# B&R Automation Studio project NAEUL004C00R13L518F00 (part 14)

#### Act_OptP0200ToP0204BypsInitConv.st
```iecst
ACTION Act_OptP0200ToP0204BypsInitConv:

	IF p_tyNtParamCurr.bProjBypsInitConvPrep THEN

		(*Display*)
		//Initializing Conveyor
		IF EDGEPOS(p_bOpsTravLifULInitConv) THEN
			fUIInRtStatOff(ADR(tyP0200OpsGen.tyBypsInitConv.tyLyr.uiRtStat));
			fUIInRtStatOff(ADR(tyP0201OpsTravLifter.tyBypsInitConv.tyLyr.uiRtStat));
			fUIInRtStatOff(ADR(tyP0202OpsMag1.tyBypsInitConv.tyLyr.uiRtStat));
			fUIInRtStatOff(ADR(tyP0203OpsMag2.tyBypsInitConv.tyLyr.uiRtStat));
			fUIInRtStatOff(ADR(tyP0204OpsMag3.tyBypsInitConv.tyLyr.uiRtStat));
			fUIInRtStatOff(ADR(tyP0206OpsMagConv1.tyBypsInitConv.tyLyr.uiRtStat));
			fUIInRtStatOff(ADR(tyP0207OpsMagConv2.tyBypsInitConv.tyLyr.uiRtStat));
		END_IF

		//Initializing Conveyor Done
		IF EDGENEG(p_bOpsTravLifULInitConv) THEN
			fUIInRtStatHide(ADR(tyP0200OpsGen.tyBypsInitConv.tyLyr.uiRtStat));
			fUIInRtStatHide(ADR(tyP0201OpsTravLifter.tyBypsInitConv.tyLyr.uiRtStat));
			fUIInRtStatHide(ADR(tyP0202OpsMag1.tyBypsInitConv.tyLyr.uiRtStat));
			fUIInRtStatHide(ADR(tyP0203OpsMag2.tyBypsInitConv.tyLyr.uiRtStat));
			fUIInRtStatHide(ADR(tyP0204OpsMag3.tyBypsInitConv.tyLyr.uiRtStat));
			fUIInRtStatHide(ADR(tyP0206OpsMagConv1.tyBypsInitConv.tyLyr.uiRtStat));
			fUIInRtStatHide(ADR(tyP0207OpsMagConv2.tyBypsInitConv.tyLyr.uiRtStat));

			bOpsBypsInitConv	:= FALSE;
		END_IF

		//Blinking Button
		IF tyP0200OpsGen.tyBypsInitConv.tyLyr.uiRtStat.0 = FALSE THEN

			fbBypsInitConvBlinkTm(IN := TRUE);

			IF fbBypsInitConvBlinkTm.Q THEN
				fbBypsInitConvBlinkTm(IN := FALSE);

				IF tyP0200OpsGen.tyBypsInitConv.tyBtnBypsInitConv.usiBitmapIdx = 0 THEN
					tyP0200OpsGen.tyBypsInitConv.tyBtnBypsInitConv.usiBitmapIdx			:= 1;
					tyP0201OpsTravLifter.tyBypsInitConv.tyBtnBypsInitConv.usiBitmapIdx	:= 1;
					tyP0202OpsMag1.tyBypsInitConv.tyBtnBypsInitConv.usiBitmapIdx		:= 1;
					tyP0203OpsMag2.tyBypsInitConv.tyBtnBypsInitConv.usiBitmapIdx		:= 1;
					tyP0204OpsMag3.tyBypsInitConv.tyBtnBypsInitConv.usiBitmapIdx		:= 1;
					tyP0206OpsMagConv1.tyBypsInitConv.tyBtnBypsInitConv.usiBitmapIdx	:= 1;
					tyP0207OpsMagConv2.tyBypsInitConv.tyBtnBypsInitConv.usiBitmapIdx	:= 1;
				ELSE
					tyP0200OpsGen.tyBypsInitConv.tyBtnBypsInitConv.usiBitmapIdx			:= 0;
					tyP0201OpsTravLifter.tyBypsInitConv.tyBtnBypsInitConv.usiBitmapIdx	:= 0;
					tyP0202OpsMag1.tyBypsInitConv.tyBtnBypsInitConv.usiBitmapIdx		:= 0;
					tyP0203OpsMag2.tyBypsInitConv.tyBtnBypsInitConv.usiBitmapIdx		:= 0;
					tyP0204OpsMag3.tyBypsInitConv.tyBtnBypsInitConv.usiBitmapIdx		:= 0;
					tyP0206OpsMagConv1.tyBypsInitConv.tyBtnBypsInitConv.usiBitmapIdx	:= 0;
					tyP0207OpsMagConv2.tyBypsInitConv.tyBtnBypsInitConv.usiBitmapIdx	:= 0;
				END_IF

			END_IF

		ELSE

			fbBypsInitConvBlinkTm(IN := FALSE);

			tyP0200OpsGen.tyBypsInitConv.tyBtnBypsInitConv.usiBitmapIdx			:= 0;
			tyP0201OpsTravLifter.tyBypsInitConv.tyBtnBypsInitConv.usiBitmapIdx	:= 0;
			tyP0202OpsMag1.tyBypsInitConv.tyBtnBypsInitConv.usiBitmapIdx		:= 0;
			tyP0203OpsMag2.tyBypsInitConv.tyBtnBypsInitConv.usiBitmapIdx		:= 0;
			tyP0204OpsMag3.tyBypsInitConv.tyBtnBypsInitConv.usiBitmapIdx		:= 0;
			tyP0206OpsMagConv1.tyBypsInitConv.tyBtnBypsInitConv.usiBitmapIdx	:= 0;
			tyP0207OpsMagConv2.tyBypsInitConv.tyBtnBypsInitConv.usiBitmapIdx	:= 0;

		END_IF

		(*Control*)
		IF tyP0200OpsGen.tyBypsInitConv.tyBtnBypsInitConv.bRtCompl OR tyP0201OpsTravLifter.tyBypsInitConv.tyBtnBypsInitConv.bRtCompl OR tyP0202OpsMag1.tyBypsInitConv.tyBtnBypsInitConv.bRtCompl OR tyP0203OpsMag2.tyBypsInitConv.tyBtnBypsInitConv.bRtCompl OR tyP0204OpsMag3.tyBypsInitConv.tyBtnBypsInitConv.bRtCompl THEN
			tyP0200OpsGen.tyBypsInitConv.tyBtnBypsInitConv.bRtCompl			:= FALSE;
			tyP0201OpsTravLifter.tyBypsInitConv.tyBtnBypsInitConv.bRtCompl	:= FALSE;
			tyP0202OpsMag1.tyBypsInitConv.tyBtnBypsInitConv.bRtCompl		:= FALSE;
			tyP0203OpsMag2.tyBypsInitConv.tyBtnBypsInitConv.bRtCompl		:= FALSE;
			tyP0204OpsMag3.tyBypsInitConv.tyBtnBypsInitConv.bRtCompl		:= FALSE;
			tyP0206OpsMagConv1.tyBypsInitConv.tyBtnBypsInitConv.bRtCompl	:= FALSE;
			tyP0207OpsMagConv2.tyBypsInitConv.tyBtnBypsInitConv.bRtCompl	:= FALSE;

			fUIInRtStatHide(ADR(tyP0200OpsGen.tyBypsInitConv.tyLyr.uiRtStat));
			fUIInRtStatHide(ADR(tyP0201OpsTravLifter.tyBypsInitConv.tyLyr.uiRtStat));
			fUIInRtStatHide(ADR(tyP0202OpsMag1.tyBypsInitConv.tyLyr.uiRtStat));
			fUIInRtStatHide(ADR(tyP0203OpsMag2.tyBypsInitConv.tyLyr.uiRtStat));
			fUIInRtStatHide(ADR(tyP0204OpsMag3.tyBypsInitConv.tyLyr.uiRtStat));
			fUIInRtStatHide(ADR(tyP0206OpsMagConv1.tyBypsInitConv.tyLyr.uiRtStat));
			fUIInRtStatHide(ADR(tyP0207OpsMagConv2.tyBypsInitConv.tyLyr.uiRtStat));

			bOpsBypsInitConv	:= TRUE;

		ELSIF tyP0200OpsGen.tyBypsInitConv.tyHotspotClose.bRtCompl OR tyP0201OpsTravLifter.tyBypsInitConv.tyHotspotClose.bRtCompl OR tyP0202OpsMag1.tyBypsInitConv.tyHotspotClose.bRtCompl OR tyP0203OpsMag2.tyBypsInitConv.tyHotspotClose.bRtCompl OR tyP0204OpsMag3.tyBypsInitConv.tyHotspotClose.bRtCompl THEN
			tyP0200OpsGen.tyBypsInitConv.tyHotspotClose.bRtCompl		:= FALSE;
			tyP0201OpsTravLifter.tyBypsInitConv.tyHotspotClose.bRtCompl	:= FALSE;
			tyP0202OpsMag1.tyBypsInitConv.tyHotspotClose.bRtCompl		:= FALSE;
			tyP0203OpsMag2.tyBypsInitConv.tyHotspotClose.bRtCompl		:= FALSE;
			tyP0204OpsMag3.tyBypsInitConv.tyHotspotClose.bRtCompl		:= FALSE;
			tyP0206OpsMagConv1.tyBypsInitConv.tyHotspotClose.bRtCompl	:= FALSE;
			tyP0207OpsMagConv2.tyBypsInitConv.tyHotspotClose.bRtCompl	:= FALSE;

			fUIInRtStatHide(ADR(tyP0200OpsGen.tyBypsInitConv.tyLyr.uiRtStat));
			fUIInRtStatHide(ADR(tyP0201OpsTravLifter.tyBypsInitConv.tyLyr.uiRtStat));
			fUIInRtStatHide(ADR(tyP0202OpsMag1.tyBypsInitConv.tyLyr.uiRtStat));
			fUIInRtStatHide(ADR(tyP0203OpsMag2.tyBypsInitConv.tyLyr.uiRtStat));
			fUIInRtStatHide(ADR(tyP0204OpsMag3.tyBypsInitConv.tyLyr.uiRtStat));
			fUIInRtStatHide(ADR(tyP0206OpsMagConv1.tyBypsInitConv.tyLyr.uiRtStat));
			fUIInRtStatHide(ADR(tyP0207OpsMagConv2.tyBypsInitConv.tyLyr.uiRtStat));

		END_IF

	END_IF

END_ACTION
```

#### Act_OptP0202ToP0204_P0003UnloadMag.st
```iecst
ACTION Act_OptP0202ToP0204_P0003UnloadMag:

	//Reset
	IF EDGEPOS(p_bOpsStatusStop) THEN
		bUnloadMag	:= FALSE;

		tyP0202OpsMag1.tyOps.tyBtnUnloadMag.bRtCompl	:= FALSE;
		tyP0203OpsMag2.tyOps.tyBtnUnloadMag.bRtCompl	:= FALSE;
		tyP0204OpsMag3.tyOps.tyBtnUnloadMag.bRtCompl	:= FALSE;

		tyP0003MMenu.tyMMenuBtn.tyBtnMnlUnload.bRtCompl := FALSE;

		p_tyC0008MsgBox ACCESS ADR(tyP0202OpsMag1.tyMsgBoxHide);
		p_tyC0008MsgBox ACCESS ADR(tyP0203OpsMag2.tyMsgBoxHide);
		p_tyC0008MsgBox ACCESS ADR(tyP0204OpsMag3.tyMsgBoxHide);

		p_tyC0008MsgBox ACCESS ADR(tyP0003MMenu.tyMsgBoxHide);
	END_IF

	//Control
	IF tyP0202OpsMag1.tyOps.tyBtnUnloadMag.bRtCompl = TRUE THEN

		IF bUnloadMag = FALSE THEN

			p_tyC0008MsgBox ACCESS ADR(tyP0202OpsMag1.tyMsgBoxUnloadAsk);

			IF tyP0202OpsMag1.tyMsgBoxUnloadAsk.tyBtnYes.bRtCompl = TRUE THEN
				tyP0202OpsMag1.tyMsgBoxUnloadAsk.tyBtnYes.bRtCompl	:= FALSE;
				tyP0202OpsMag1.tyMsgBoxUnloadAsk.tyBtnYes.bValue	:= FALSE;

				p_tyC0008MsgBox ACCESS ADR(tyP0202OpsMag1.tyMsgBoxHide);

				bUnloadMag	:= TRUE;

				tyP0202OpsMag1.tyOps.tyBtnUnloadMag.bRtCompl	:= FALSE;

			ELSIF tyP0202OpsMag1.tyMsgBoxUnloadAsk.tyBtnNo.bRtCompl = TRUE THEN
				tyP0202OpsMag1.tyMsgBoxUnloadAsk.tyBtnNo.bRtCompl	:= FALSE;
				tyP0202OpsMag1.tyMsgBoxUnloadAsk.tyBtnNo.bValue		:= FALSE;

				p_tyC0008MsgBox ACCESS ADR(tyP0202OpsMag1.tyMsgBoxHide);

				tyP0202OpsMag1.tyOps.tyBtnUnloadMag.bRtCompl	:= FALSE;

			END_IF

		ELSE

			p_tyC0008MsgBox ACCESS ADR(tyP0202OpsMag1.tyMsgBoxResumeAsk);

			IF tyP0202OpsMag1.tyMsgBoxResumeAsk.tyBtnYes.bRtCompl = TRUE THEN
				tyP0202OpsMag1.tyMsgBoxResumeAsk.tyBtnYes.bRtCompl	:= FALSE;
				tyP0202OpsMag1.tyMsgBoxResumeAsk.tyBtnYes.bValue	:= FALSE;

				p_tyC0008MsgBox ACCESS ADR(tyP0202OpsMag1.tyMsgBoxHide);

				bUnloadMag	:= FALSE;

				tyP0202OpsMag1.tyOps.tyBtnUnloadMag.bRtCompl	:= FALSE;

			ELSIF tyP0202OpsMag1.tyMsgBoxResumeAsk.tyBtnNo.bRtCompl = TRUE THEN
				tyP0202OpsMag1.tyMsgBoxResumeAsk.tyBtnNo.bRtCompl	:= FALSE;
				tyP0202OpsMag1.tyMsgBoxResumeAsk.tyBtnNo.bValue		:= FALSE;

				p_tyC0008MsgBox ACCESS ADR(tyP0202OpsMag1.tyMsgBoxHide);

				tyP0202OpsMag1.tyOps.tyBtnUnloadMag.bRtCompl	:= FALSE;

			END_IF

		END_IF

	ELSIF tyP0203OpsMag2.tyOps.tyBtnUnloadMag.bRtCompl = TRUE THEN

		IF bUnloadMag = FALSE THEN

			p_tyC0008MsgBox ACCESS ADR(tyP0203OpsMag2.tyMsgBoxUnloadAsk);

			IF tyP0203OpsMag2.tyMsgBoxUnloadAsk.tyBtnYes.bRtCompl = TRUE THEN
				tyP0203OpsMag2.tyMsgBoxUnloadAsk.tyBtnYes.bRtCompl	:= FALSE;
				tyP0203OpsMag2.tyMsgBoxUnloadAsk.tyBtnYes.bValue	:= FALSE;

				p_tyC0008MsgBox ACCESS ADR(tyP0203OpsMag2.tyMsgBoxHide);

				bUnloadMag	:= TRUE;

				tyP0203OpsMag2.tyOps.tyBtnUnloadMag.bRtCompl	:= FALSE;

			ELSIF tyP0203OpsMag2.tyMsgBoxUnloadAsk.tyBtnNo.bRtCompl = TRUE THEN
				tyP0203OpsMag2.tyMsgBoxUnloadAsk.tyBtnNo.bRtCompl	:= FALSE;
				tyP0203OpsMag2.tyMsgBoxUnloadAsk.tyBtnNo.bValue		:= FALSE;

				p_tyC0008MsgBox ACCESS ADR(tyP0203OpsMag2.tyMsgBoxHide);

				tyP0203OpsMag2.tyOps.tyBtnUnloadMag.bRtCompl	:= FALSE;

			END_IF

		ELSE

			p_tyC0008MsgBox ACCESS ADR(tyP0203OpsMag2.tyMsgBoxResumeAsk);

			IF tyP0203OpsMag2.tyMsgBoxResumeAsk.tyBtnYes.bRtCompl = TRUE THEN
				tyP0203OpsMag2.tyMsgBoxResumeAsk.tyBtnYes.bRtCompl	:= FALSE;
				tyP0203OpsMag2.tyMsgBoxResumeAsk.tyBtnYes.bValue	:= FALSE;

				p_tyC0008MsgBox ACCESS ADR(tyP0203OpsMag2.tyMsgBoxHide);

				bUnloadMag	:= FALSE;

				tyP0203OpsMag2.tyOps.tyBtnUnloadMag.bRtCompl	:= FALSE;

			ELSIF tyP0203OpsMag2.tyMsgBoxResumeAsk.tyBtnNo.bRtCompl = TRUE THEN
				tyP0203OpsMag2.tyMsgBoxResumeAsk.tyBtnNo.bRtCompl	:= FALSE;
				tyP0203OpsMag2.tyMsgBoxResumeAsk.tyBtnNo.bValue		:= FALSE;

				p_tyC0008MsgBox ACCESS ADR(tyP0203OpsMag2.tyMsgBoxHide);

				tyP0203OpsMag2.tyOps.tyBtnUnloadMag.bRtCompl	:= FALSE;

			END_IF

		END_IF

	ELSIF tyP0204OpsMag3.tyOps.tyBtnUnloadMag.bRtCompl = TRUE THEN

		IF bUnloadMag = FALSE THEN

			p_tyC0008MsgBox ACCESS ADR(tyP0204OpsMag3.tyMsgBoxUnloadAsk);

			IF tyP0204OpsMag3.tyMsgBoxUnloadAsk.tyBtnYes.bRtCompl = TRUE THEN
				tyP0204OpsMag3.tyMsgBoxUnloadAsk.tyBtnYes.bRtCompl	:= FALSE;
				tyP0204OpsMag3.tyMsgBoxUnloadAsk.tyBtnYes.bValue	:= FALSE;

				p_tyC0008MsgBox ACCESS ADR(tyP0204OpsMag3.tyMsgBoxHide);

				bUnloadMag	:= TRUE;

				tyP0204OpsMag3.tyOps.tyBtnUnloadMag.bRtCompl	:= FALSE;

			ELSIF tyP0204OpsMag3.tyMsgBoxUnloadAsk.tyBtnNo.bRtCompl = TRUE THEN
				tyP0204OpsMag3.tyMsgBoxUnloadAsk.tyBtnNo.bRtCompl	:= FALSE;
				tyP0204OpsMag3.tyMsgBoxUnloadAsk.tyBtnNo.bValue		:= FALSE;

				p_tyC0008MsgBox ACCESS ADR(tyP0204OpsMag3.tyMsgBoxHide);

				tyP0204OpsMag3.tyOps.tyBtnUnloadMag.bRtCompl	:= FALSE;

			END_IF

		ELSE

			p_tyC0008MsgBox ACCESS ADR(tyP0204OpsMag3.tyMsgBoxResumeAsk);

			IF tyP0204OpsMag3.tyMsgBoxResumeAsk.tyBtnYes.bRtCompl = TRUE THEN
				tyP0204OpsMag3.tyMsgBoxResumeAsk.tyBtnYes.bRtCompl	:= FALSE;
				tyP0204OpsMag3.tyMsgBoxResumeAsk.tyBtnYes.bValue	:= FALSE;

				p_tyC0008MsgBox ACCESS ADR(tyP0204OpsMag3.tyMsgBoxHide);

				bUnloadMag	:= FALSE;

				tyP0204OpsMag3.tyOps.tyBtnUnloadMag.bRtCompl	:= FALSE;

			ELSIF tyP0204OpsMag3.tyMsgBoxResumeAsk.tyBtnNo.bRtCompl = TRUE THEN
				tyP0204OpsMag3.tyMsgBoxResumeAsk.tyBtnNo.bRtCompl	:= FALSE;
				tyP0204OpsMag3.tyMsgBoxResumeAsk.tyBtnNo.bValue		:= FALSE;

				p_tyC0008MsgBox ACCESS ADR(tyP0204OpsMag3.tyMsgBoxHide);

				tyP0204OpsMag3.tyOps.tyBtnUnloadMag.bRtCompl	:= FALSE;

			END_IF

		END_IF
		////////
	ELSIF tyP0003MMenu.tyMMenuBtn.tyBtnMnlUnload.bRtCompl = TRUE THEN

		IF bUnloadMag = FALSE THEN

			p_tyC0008MsgBox ACCESS ADR(tyP0003MMenu.tyMsgBoxUnloadAsk);

			IF tyP0003MMenu.tyMsgBoxUnloadAsk.tyBtnYes.bRtCompl = TRUE THEN
				tyP0003MMenu.tyMsgBoxUnloadAsk.tyBtnYes.bRtCompl	:= FALSE;
				tyP0003MMenu.tyMsgBoxUnloadAsk.tyBtnYes.bValue	:= FALSE;

				p_tyC0008MsgBox ACCESS ADR(tyP0003MMenu.tyMsgBoxHide);

				bUnloadMag	:= TRUE;

				tyP0003MMenu.tyMMenuBtn.tyBtnMnlUnload.bRtCompl	:= FALSE;

			ELSIF tyP0003MMenu.tyMsgBoxUnloadAsk.tyBtnNo.bRtCompl = TRUE THEN
				tyP0003MMenu.tyMsgBoxUnloadAsk.tyBtnNo.bRtCompl	:= FALSE;
				tyP0003MMenu.tyMsgBoxUnloadAsk.tyBtnNo.bValue		:= FALSE;

				p_tyC0008MsgBox ACCESS ADR(tyP0003MMenu.tyMsgBoxHide);

				tyP0003MMenu.tyMMenuBtn.tyBtnMnlUnload.bRtCompl	:= FALSE;

			END_IF

		ELSE

			p_tyC0008MsgBox ACCESS ADR(tyP0003MMenu.tyMsgBoxResumeAsk);

			IF tyP0003MMenu.tyMsgBoxResumeAsk.tyBtnYes.bRtCompl = TRUE THEN
				tyP0003MMenu.tyMsgBoxResumeAsk.tyBtnYes.bRtCompl	:= FALSE;
				tyP0003MMenu.tyMsgBoxResumeAsk.tyBtnYes.bValue	:= FALSE;

				p_tyC0008MsgBox ACCESS ADR(tyP0003MMenu.tyMsgBoxHide);

				bUnloadMag	:= FALSE;

				tyP0003MMenu.tyMMenuBtn.tyBtnMnlUnload.bRtCompl	:= FALSE;

			ELSIF tyP0003MMenu.tyMsgBoxResumeAsk.tyBtnNo.bRtCompl = TRUE THEN
				tyP0003MMenu.tyMsgBoxResumeAsk.tyBtnNo.bRtCompl	:= FALSE;
				tyP0003MMenu.tyMsgBoxResumeAsk.tyBtnNo.bValue		:= FALSE;

				p_tyC0008MsgBox ACCESS ADR(tyP0003MMenu.tyMsgBoxHide);

				tyP0003MMenu.tyMMenuBtn.tyBtnMnlUnload.bRtCompl	:= FALSE;

			END_IF

		END_IF

	END_IF

	//Display
	tyP0202OpsMag1.tyOps.tyBtnUnloadMag.bRtLk	:= p_bOpsStatusStop = FALSE AND bUnloadMag AND NOT p_bOpsLifMagULUnloading;
	tyP0203OpsMag2.tyOps.tyBtnUnloadMag.bRtLk	:= p_bOpsStatusStop = FALSE AND bUnloadMag AND NOT p_bOpsLifMagULUnloading;
	tyP0204OpsMag3.tyOps.tyBtnUnloadMag.bRtLk	:= p_bOpsStatusStop = FALSE AND bUnloadMag AND NOT p_bOpsLifMagULUnloading;
	tyP0003MMenu.tyMMenuBtn.tyBtnMnlUnload.bRtLk := p_bOpsStatusStop = FALSE AND bUnloadMag AND NOT p_bOpsLifMagULUnloading;

	IF p_bOpsStatusStop = FALSE AND p_bOpsLifMagULUnloading = TRUE THEN
		tyP0202OpsMag1.tyOps.tyBtnUnloadMag.usiTxtIdx	:= 1;
		tyP0203OpsMag2.tyOps.tyBtnUnloadMag.usiTxtIdx	:= 1;
		tyP0204OpsMag3.tyOps.tyBtnUnloadMag.usiTxtIdx	:= 1;
		tyP0003MMenu.tyMMenuBtn.tyBtnMnlUnload.usiTxtIdx	:= 30;
	ELSE
		tyP0202OpsMag1.tyOps.tyBtnUnloadMag.usiTxtIdx	:= 0;
		tyP0203OpsMag2.tyOps.tyBtnUnloadMag.usiTxtIdx	:= 0;
		tyP0204OpsMag3.tyOps.tyBtnUnloadMag.usiTxtIdx	:= 0;
		tyP0003MMenu.tyMMenuBtn.tyBtnMnlUnload.usiTxtIdx	:= 5;
	END_IF

	IF p_bOpsStatusStop = FALSE AND bUnloadMag = TRUE AND p_bOpsLifMagULUnloading = TRUE THEN

		fbUnloadBlinkTm(IN := TRUE);

		IF fbUnloadBlinkTm.Q = TRUE THEN
			fbUnloadBlinkTm(IN := FALSE);

			IF tyP0202OpsMag1.tyOps.tyBitmapUnloadMag.usiValueIdx = 0 THEN
				tyP0202OpsMag1.tyOps.tyBitmapUnloadMag.usiValueIdx	:= 3;
				tyP0203OpsMag2.tyOps.tyBitmapUnloadMag.usiValueIdx	:= 3;
				tyP0204OpsMag3.tyOps.tyBitmapUnloadMag.usiValueIdx	:= 3;

				tyP0003MMenu.tyMMenuBtn.tyBtnMnlUnload.usiBitmapIdx    := 4; //Yellow
			ELSE
				tyP0202OpsMag1.tyOps.tyBitmapUnloadMag.usiValueIdx	:= 0;
				tyP0203OpsMag2.tyOps.tyBitmapUnloadMag.usiValueIdx	:= 0;
				tyP0204OpsMag3.tyOps.tyBitmapUnloadMag.usiValueIdx	:= 0;

				tyP0003MMenu.tyMMenuBtn.tyBtnMnlUnload.usiBitmapIdx    := 0; //Silver
			END_IF

		END_IF

	ELSIF p_bOpsStatusStop = FALSE AND bUnloadMag = TRUE THEN

		fbUnloadBlinkTm(IN := FALSE);

		tyP0202OpsMag1.tyOps.tyBitmapUnloadMag.usiValueIdx	:= 1;
		tyP0203OpsMag2.tyOps.tyBitmapUnloadMag.usiValueIdx	:= 1;
		tyP0204OpsMag3.tyOps.tyBitmapUnloadMag.usiValueIdx	:= 1;

		tyP0003MMenu.tyMMenuBtn.tyBtnMnlUnload.usiBitmapIdx    := 1; //Green

	ELSE

		fbUnloadBlinkTm(IN := FALSE);

		tyP0202OpsMag1.tyOps.tyBitmapUnloadMag.usiValueIdx	:= 0;
		tyP0203OpsMag2.tyOps.tyBitmapUnloadMag.usiValueIdx	:= 0;
		tyP0204OpsMag3.tyOps.tyBitmapUnloadMag.usiValueIdx	:= 0;

		tyP0003MMenu.tyMMenuBtn.tyBtnMnlUnload.usiBitmapIdx    := 0;

	END_IF

	//Mask
	IF p_tyNtParamCurr.bProjLifterMagPlatform THEN
		IF p_bOpsStatusStop
			OR (p_bOpsTravLifMov AND p_bPshrConvHvBrd AND NOT(p_bOutShutterRetracted))
			THEN //p_bOpsLifMagULLifMov

			fUIInRtStatOff(ADR(tyP0202OpsMag1.tyOps.tyBtnUnloadMag.uiMaskRtStat));
			fUIInRtStatOff(ADR(tyP0203OpsMag2.tyOps.tyBtnUnloadMag.uiMaskRtStat));
			fUIInRtStatOff(ADR(tyP0204OpsMag3.tyOps.tyBtnUnloadMag.uiMaskRtStat));
			fUIInRtStatOff(ADR(tyP0003MMenu.tyMMenuBtn.tyBtnMnlUnload.uiMaskRtStat));
		ELSE
			fUIInRtStatHide(ADR(tyP0202OpsMag1.tyOps.tyBtnUnloadMag.uiMaskRtStat));
			fUIInRtStatHide(ADR(tyP0203OpsMag2.tyOps.tyBtnUnloadMag.uiMaskRtStat));
			fUIInRtStatHide(ADR(tyP0204OpsMag3.tyOps.tyBtnUnloadMag.uiMaskRtStat));
			fUIInRtStatHide(ADR(tyP0003MMenu.tyMMenuBtn.tyBtnMnlUnload.uiMaskRtStat));
		END_IF
	END_IF
END_ACTION
```

#### Act_EntP0300Disp.st
```iecst
ACTION Act_EntP0300Disp:

	//Access Addres
	p_tyC0005Main ACCESS ADR(tyCommon.tyMain);

	p_tyC0007Notif ACCESS ADR(tyCommon.tyNotif);

	p_tyC0008MsgBox ACCESS ADR(tyP0300McInfo.tyMsgBoxHide);

	p_tyC0009Info ACCESS ADR(tyCommon.tyInfo);

	p_tyP0300McInfo ACCESS ADR(tyP0300McInfo.tyMcInfo);

	//Display
	//Machine Name
	tyP0300McInfo.tyMcInfo.tyStringMcNm.sValue	:= p_tyMcParamCurr.sMcNm;

END_ACTION
```

#### Act_EntP0400Disp.st
```iecst
ACTION Act_EntP0400Disp:

	//Access Addres
	p_tyC0005Main ACCESS ADR(tyCommon.tyMain);

	p_tyC0007Notif ACCESS ADR(tyCommon.tyNotif);

	p_tyC0008MsgBox ACCESS ADR(tyP0400ProdSel.tyMsgBoxHide);

	p_tyC0009Info ACCESS ADR(tyCommon.tyInfo);

	p_tyC0011RcpPopUp ACCESS ADR(tyP0400ProdSel.tyRcpPopUp);

	p_tyP0400ProdSel ACCESS ADR(tyP0400ProdSel.tyProdSel);
	p_tyP0400RcpDet ACCESS ADR(tyP0400ProdSel.tyRcpDet);

	//Display
	tyP0400ProdSel.tyProdSel.tyBtnSort.bRtCompl			:= FALSE;
	tyP0400ProdSel.tyProdSel.tyBtnSort.bValue			:= FALSE;
	tyP0400ProdSel.tyProdSel.tyStringSearch.bRtCompl			:= TRUE;
	fUIInRtStatHide(ADR(tyP0400ProdSel.tyRcpDet.tyLyr.uiRtStat));

	fUIInRtStatHide(ADR(tyP0400ProdSel.tyRcpPopUp.tyLyr.uiRtStat)); // Hide Pop Up Layer

	//Long Board
	tyP0400ProdSel.tyProdSel.tyBtnLongBrd.uiRtStat.0			:= NOT(p_tyNtParamCurr.bProjLongBrdPrep AND p_tyMcParamCurr.bLongBrdEn);
	tyP0400ProdSel.tyRcpDet.tyBtnLongBrd.uiRtStat.0				:= NOT(p_tyNtParamCurr.bProjLongBrdPrep AND p_tyMcParamCurr.bLongBrdEn);

	//Gap Between Board
	tyP0400ProdSel.tyProdSel.tyBtnGapBetBrds.uiRtStat.0			:= NOT p_tyMcParamCurr.bGapBwtnBrdEn;
	tyP0400ProdSel.tyRcpDet.tyBtnGapBetBrd.uiRtStat.0			:= NOT p_tyMcParamCurr.bGapBwtnBrdEn;

	//Oven Info
	tyP0400ProdSel.tyProdSel.tyNumMinReqFreeBffr.uiRtStat.0		:= NOT(p_tyNtParamCurr.bOvenInfoPrep AND NOT(p_tyNtParamCurr.bOvenInfoExtdPrep AND p_tyMcParamCurr.bExtdOvenEn));
	tyP0400ProdSel.tyProdSel.tyTxtMinReqFreeBffr.uiRtStat.0		:= NOT(p_tyNtParamCurr.bOvenInfoPrep AND NOT(p_tyNtParamCurr.bOvenInfoExtdPrep AND p_tyMcParamCurr.bExtdOvenEn));
	tyP0400ProdSel.tyRcpDet.tyNumMinReqFreeBffr.uiRtStat.0		:= NOT(p_tyNtParamCurr.bOvenInfoPrep AND NOT(p_tyNtParamCurr.bOvenInfoExtdPrep AND p_tyMcParamCurr.bExtdOvenEn));
	tyP0400ProdSel.tyRcpDet.tyTxtMinReqFreeBffr.uiRtStat.0		:= NOT(p_tyNtParamCurr.bOvenInfoPrep AND NOT(p_tyNtParamCurr.bOvenInfoExtdPrep AND p_tyMcParamCurr.bExtdOvenEn));

	//Product Selection
	tyP0400ProdSel.tyProdSel.tyStringRecipeNm.sValue			:= p_tyProdRcpCurrRcp0.sRcpNm;
	tyP0400ProdSel.tyProdSel.tyNumProdWidth.diValue				:= p_tyProdRcpCurrRcp0.diWidthInUM;
	tyP0400ProdSel.tyProdSel.tyNumMaxSlt.diValue				:= p_tyProdRcpCurrRcp0.diMaxSltValue;
	tyP0400ProdSel.tyProdSel.tyNumMinSlt.diValue				:= p_tyProdRcpCurrRcp0.diMinSltValue;
	tyP0400ProdSel.tyProdSel.tyNumPitch.diValue					:= p_tyProdRcpCurrRcp0.diPitch;
	tyP0400ProdSel.tyProdSel.tyNumBrdPerSlt.diValue				:= p_tyProdRcpCurrRcp0.diBrdPerSlt;
	tyP0400ProdSel.tyProdSel.tyBtnToptoBtm.bValue				:= p_tyProdRcpCurrRcp0.bTopToBtm;
	tyP0400ProdSel.tyProdSel.tyBtnGapBetBrds.bValue				:= p_tyProdRcpCurrRcp0.bGapBwtnBrd;
	tyP0400ProdSel.tyProdSel.tyBtnLongBrd.bValue				:= p_tyProdRcpCurrRcp0.bLongBrd;
	tyP0400ProdSel.tyProdSel.tyTxtMcMode.usiValueIdx			:= p_tyProdRcpCurrRcp0.usiMcMod;
	tyP0400ProdSel.tyProdSel.tyNumMinReqFreeBffr.diValue		:= p_tyProdRcpCurrRcp0.diMinReqFreeBffr;
	tyP0400ProdSel.tyProdSel.tyNumProdWidth2.diValue			:= p_tyProdRcpCurrRcp0.diWidthInUM2;
	tyP0400ProdSel.tyProdSel.tyNumMtrPshrExtSpd.diValue			:= p_tyProdRcpCurrRcp0.diMtrPshrExtSpd;
	tyP0400ProdSel.tyProdSel.tyNumMtrPshrExtTorq.diValue		:= p_tyProdRcpCurrRcp0.diMtrPshrExtTorq;
	tyP0400ProdSel.tyProdSel.tyNumPshrOffset.diValue			:= p_tyProdRcpCurrRcp0.diPshrOffset;

END_ACTION
```

#### Act_OptP0400Search.st
```iecst
ACTION Act_OptP0400Search:

	IF tyP0400ProdSel.tyProdSel.tyStringSearch.bRtCompl = TRUE THEN	//Search Input Valid
		IF tyP0400ProdSel.tyProdSel.tyStringSearch.sValue = '' THEN
			FOR i := 1 TO c_uiP0400TableSize DO
				tyP0400ProdSel.tyProdSel.tyTableRecipe.a_tyStringDataCol0[i].sValue	:= UINT_TO_STRING(tyP0400Table.uiTablePos + i - 1);
				tyP0400ProdSel.tyProdSel.tyTableRecipe.a_tyStringDataCol1[i].sValue	:= p_tyProdRcpCurrList[tyP0400Table.uiTablePos + i - 1].sRcpNm;
				tyP0400ProdSel.tyProdSel.tyTableRecipe.a_tyStringDataCol2[i].sValue	:= p_tyProdRcpCurrList[tyP0400Table.uiTablePos + i - 1].sDisplayInfo;
			END_FOR

			tyP0400ProdSel.tyProdSel.tyStringSearch.bRtCompl	:= FALSE;

			IF tyP0400ProdSel.tyProdSel.tyBtnSort.bValue THEN
				bFilterSortP0400	:= TRUE;
			END_IF

		ELSE
			//Mask
			tyP0400ProdSel.tyProdSel.tyTableRecipe.uiMaskRtStat.0	:= FALSE;

			sProdRcpSearch	:= tyP0400ProdSel.tyProdSel.tyStringSearch.sValue;

			eProdRcpAct	:= ProdRcpActFilter;

			IF p_eProdRcpStat = ProdRcpActFilter AND p_eProdRcpStatus = Done THEN
				eProdRcpAct		:= ProdRcpActIdle;

				FOR i := 1 TO c_uiP1040TableSize DO
					tyP0400ProdSel.tyProdSel.tyTableRecipe.a_tyStringDataCol0[i].sValue	:= UINT_TO_STRING(tyP0400Table.uiTablePos + i - 1);
					tyP0400ProdSel.tyProdSel.tyTableRecipe.a_tyStringDataCol1[i].sValue	:= p_tyProdRcpFilterList[tyP0400Table.uiTablePos + i - 1].sRcpNm;
					tyP0400ProdSel.tyProdSel.tyTableRecipe.a_tyStringDataCol2[i].sValue	:= p_tyProdRcpFilterList[tyP0400Table.uiTablePos + i - 1].sDisplayInfo;
				END_FOR

				//Unmask
				tyP0400ProdSel.tyProdSel.tyTableRecipe.uiMaskRtStat.0	:= TRUE;

				tyP0400ProdSel.tyProdSel.tyStringSearch.bRtCompl		:= FALSE;

				IF tyP0400ProdSel.tyProdSel.tyBtnSort.bValue THEN
					bFilterSortP0400	:= TRUE;
				END_IF

			ELSIF p_eProdRcpStatus = Error THEN
				FOR i := 1 TO c_uiP0400TableSize DO
					tyP0400ProdSel.tyProdSel.tyTableRecipe.a_tyStringDataCol0[i].sValue		:= UINT_TO_STRING(tyP0400Table.uiTablePos + i - 1);
					tyP0400ProdSel.tyProdSel.tyTableRecipe.a_tyStringDataCol1[i].sValue		:= '';
					tyP0400ProdSel.tyProdSel.tyTableRecipe.a_tyStringDataCol2[i].sValue		:= '';
				END_FOR

				p_tyC0008MsgBox ACCESS ADR (tyP0400ProdSel.tyMsgBoxListErr);

				IF tyP0400ProdSel.tyMsgBoxListErr.tyBtnNo.bRtCompl = TRUE THEN
					tyP0400ProdSel.tyMsgBoxListErr.tyBtnNo.bRtCompl 		:= TRUE;
					tyP0400ProdSel.tyMsgBoxListErr.tyBtnNo.bValue			:= TRUE;

					p_tyC0008MsgBox ACCESS ADR (tyP0400ProdSel.tyMsgBoxHide);

					//Unmask
					tyP0400ProdSel.tyProdSel.tyTableRecipe.uiMaskRtStat.0	:= TRUE;

					//Reset
					tyP0400ProdSel.tyProdSel.tyStringSearch.bRtCompl		:= FALSE;
				END_IF
			END_IF
		END_IF
	END_IF

END_ACTION
```

#### Act_OptP0400Load.st
```iecst
ACTION Act_OptP0400Load:

	IF tyP0400ProdSel.tyProdSel.tyBtnLoad.bRtCompl = TRUE THEN

		IF usiSelProdRcpStep = 0 THEN
			//Message Confirmation Ask - Load Product Recipe
			//Mask
			tyP0400ProdSel.tyProdSel.tyTableRecipe.uiMaskRtStat		:= FALSE;
			tyP0400ProdSel.tyProdSel.tyStringSearch.uiMaskRtStat	:= FALSE;

			p_tyC0008MsgBox ACCESS ADR(tyP0400ProdSel.tyMsgBoxSelRcpAsk);

			IF tyP0400ProdSel.tyMsgBoxSelRcpAsk.tyBtnYes.bRtCompl = TRUE THEN
				tyP0400ProdSel.tyMsgBoxSelRcpAsk.tyBtnYes.bRtCompl	:= FALSE;
				tyP0400ProdSel.tyMsgBoxSelRcpAsk.tyBtnYes.bValue	:= FALSE;

				p_tyC0008MsgBox ACCESS ADR(tyP0400ProdSel.tyMsgBoxHide);

				usiSelProdRcpStep	:= 1;

			ELSIF tyP0400ProdSel.tyMsgBoxSelRcpAsk.tyBtnNo.bRtCompl = TRUE THEN
				tyP0400ProdSel.tyMsgBoxSelRcpAsk.tyBtnNo.bRtCompl	:= FALSE;
				tyP0400ProdSel.tyMsgBoxSelRcpAsk.tyBtnNo.bValue		:= FALSE;

				p_tyC0008MsgBox ACCESS ADR(tyP0400ProdSel.tyMsgBoxHide);

				usiSelProdRcpStep	:= 99;

			END_IF

		ELSIF usiSelProdRcpStep = 1 THEN
			//Load Product Recipe
			tyProdRcpInfoIn.sRcpNm		:= tyP0400ProdSel.tyProdSel.tyTableRecipe.a_tyStringDataCol1[tyP0400Table.uiSelectedRow].sValue;

			eProdRcpAct					:= ProdRcpActLoadRcp;

			IF p_eProdRcpStat = ProdRcpActLoadRcp AND p_eProdRcpStatus = Done THEN
				eProdRcpAct				:= ProdRcpActIdle;

				IF p_bProdRcpNmEmpty = TRUE AND p_bProdRcpNmNotExist = TRUE THEN
					usiSelProdRcpStep	:= 2;
				ELSE
					//Update UI Current Recipe
					tyP0400ProdSel.tyProdSel.tyStringRecipeNm.sValue		:= p_tyProdRcpCurrRcp0.sRcpNm;
					tyP0400ProdSel.tyProdSel.tyNumProdWidth.diValue			:= p_tyProdRcpCurrRcp0.diWidthInUM;
					tyP0400ProdSel.tyProdSel.tyNumMinSlt.diValue			:= p_tyProdRcpCurrRcp0.diMinSltValue;
					tyP0400ProdSel.tyProdSel.tyNumMaxSlt.diValue			:= p_tyProdRcpCurrRcp0.diMaxSltValue;
					tyP0400ProdSel.tyProdSel.tyNumPitch.diValue				:= p_tyProdRcpCurrRcp0.diPitch;
					tyP0400ProdSel.tyProdSel.tyBtnToptoBtm.bValue			:= p_tyProdRcpCurrRcp0.bTopToBtm;
					tyP0400ProdSel.tyProdSel.tyBtnGapBetBrds.bValue			:= p_tyProdRcpCurrRcp0.bGapBwtnBrd;
					tyP0400ProdSel.tyProdSel.tyBtnLongBrd.bValue			:= p_tyProdRcpCurrRcp0.bLongBrd;
					tyP0400ProdSel.tyProdSel.tyNumBrdPerSlt.diValue			:= p_tyProdRcpCurrRcp0.diBrdPerSlt;
					tyP0400ProdSel.tyProdSel.tyTxtMcMode.usiValueIdx		:= p_tyProdRcpCurrRcp0.usiMcMod;
					tyP0400ProdSel.tyProdSel.tyNumMinReqFreeBffr.diValue	:= p_tyProdRcpCurrRcp0.diMinReqFreeBffr;
					tyP0400ProdSel.tyProdSel.tyNumProdWidth2.diValue		:= p_tyProdRcpCurrRcp0.diWidthInUM2;
					tyP0400ProdSel.tyProdSel.tyNumMtrPshrExtSpd.diValue		:= p_tyProdRcpCurrRcp0.diMtrPshrExtSpd;
					tyP0400ProdSel.tyProdSel.tyNumMtrPshrExtTorq.diValue	:= p_tyProdRcpCurrRcp0.diMtrPshrExtTorq;
					tyP0400ProdSel.tyProdSel.tyNumPshrOffset.diValue		:= p_tyProdRcpCurrRcp0.diPshrOffset;

					tyProdRcpCurrRcpWr	:= p_tyProdRcpCurrRcp0;

					IF ((NOT p_tyNtParamCurr.bLFUsrSetPrep AND p_tyNtParamCurr.bLeaderMc) OR (p_tyNtParamCurr.bLFUsrSetPrep AND p_tyMcParamCurr.bLFLeaderMc)) AND p_tyNtParamCurr.bLFPrep AND p_tyMcParamCurr.bLFEn AND p_tyUsrMgmtCurrAccessRgt.bLFCtrl THEN
						usiSelProdRcpStep	:= 98;
					ELSE
						usiSelProdRcpStep	:= 99;
					END_IF

				END_IF

			ELSIF p_eProdRcpStatus = Error THEN

				usiSelProdRcpStep	:= 99;

			END_IF

		ELSIF usiSelProdRcpStep = 2 THEN
			//Message Name Not Found
			p_tyC0008MsgBox ACCESS ADR(tyP0400ProdSel.tyMsgBoxSelRcpNoNm);

			IF tyP0400ProdSel.tyMsgBoxSelRcpNoNm.tyBtnNo.bRtCompl = TRUE THEN
				tyP0400ProdSel.tyMsgBoxSelRcpNoNm.tyBtnNo.bRtCompl	:= FALSE;
				tyP0400ProdSel.tyMsgBoxSelRcpNoNm.tyBtnNo.bValue	:= FALSE;

				p_tyC0008MsgBox ACCESS ADR(tyP0400ProdSel.tyMsgBoxHide);

				usiSelProdRcpStep	:= 99;

			END_IF

		ELSIF usiSelProdRcpStep = 98 THEN
			//Message Confirmation Ask - Go To Leader Follower Control Page
			p_tyC0008MsgBox ACCESS ADR(tyP0400ProdSel.tyMsgBoxGoToLFCtrlAsk);

			IF tyP0400ProdSel.tyMsgBoxGoToLFCtrlAsk.tyBtnYes.bRtCompl = TRUE THEN
				tyP0400ProdSel.tyMsgBoxGoToLFCtrlAsk.tyBtnYes.bRtCompl	:= FALSE;
				tyP0400ProdSel.tyMsgBoxGoToLFCtrlAsk.tyBtnYes.bValue	:= FALSE;

				p_tyC0008MsgBox ACCESS ADR(tyP0400ProdSel.tyMsgBoxHide);

				eChgPage	:= UIP0700LFCtrl;

				tyCommon.tyMain.tyBtnStart.bRtCompl	:= TRUE;

				//Complete
				//Unmask
				tyP0400ProdSel.tyProdSel.tyTableRecipe.uiMaskRtStat		:= TRUE;
				tyP0400ProdSel.tyProdSel.tyStringSearch.uiMaskRtStat	:= TRUE;

				//Reset
				tyP0400ProdSel.tyProdSel.tyBtnLoad.bRtCompl	:= FALSE;
				tyP0400ProdSel.tyProdSel.tyBtnLoad.bValue	:= FALSE;

				usiSelProdRcpStep	:= 0;

			ELSIF tyP0400ProdSel.tyMsgBoxGoToLFCtrlAsk.tyBtnNo.bRtCompl = TRUE THEN
				tyP0400ProdSel.tyMsgBoxGoToLFCtrlAsk.tyBtnNo.bRtCompl	:= FALSE;
				tyP0400ProdSel.tyMsgBoxGoToLFCtrlAsk.tyBtnNo.bValue		:= FALSE;

				p_tyC0008MsgBox ACCESS ADR(tyP0400ProdSel.tyMsgBoxHide);

				usiSelProdRcpStep	:= 99;

			END_IF

		ELSIF usiSelProdRcpStep = 99 THEN
			//Complete
			//Unmask
			tyP0400ProdSel.tyProdSel.tyTableRecipe.uiMaskRtStat		:= TRUE;
			tyP0400ProdSel.tyProdSel.tyStringSearch.uiMaskRtStat	:= TRUE;

			//Reset
			tyP0400ProdSel.tyProdSel.tyBtnLoad.bRtCompl				:= FALSE;
			tyP0400ProdSel.tyProdSel.tyBtnLoad.bValue				:= FALSE;

			usiSelProdRcpStep	:= 0;

		END_IF

	END_IF

END_ACTION
```

#### Act_OptP0400Preview.st
```iecst
ACTION Act_OptP0400Preview:

	IF tyP0400ProdSel.tyProdSel.tyBtnPreview.bRtCompl = TRUE THEN

		tyProdRcpInfoIn.sRcpNm	:= tyP0400ProdSel.tyProdSel.tyTableRecipe.a_tyStringDataCol1[tyP0400Table.uiSelectedRow].sValue;

		eProdRcpAct	:= ProdRcpActGetInfo;

		IF	p_eProdRcpStat = ProdRcpActGetInfo AND p_eProdRcpStatus = Done THEN
			eProdRcpAct	:= ProdRcpActIdle;

			IF p_bProdRcpNmEmpty = TRUE AND p_bProdRcpNmNotExist = TRUE THEN
				tyP0400ProdSel.tyRcpDet.tyStringRecipeNm.sValue			:= '';
				tyP0400ProdSel.tyRcpDet.tyNumProdWidth.diValue			:= 100000;
				tyP0400ProdSel.tyRcpDet.tyNumProdWidth2.diValue			:= 100000;
				tyP0400ProdSel.tyRcpDet.tyTxtMcMode.usiValueIdx			:= p_tyMcParamCurr.usiDefaultMcMod;
				tyP0400ProdSel.tyRcpDet.tyNumFirstSlt.diValue			:= 0;
				tyP0400ProdSel.tyRcpDet.tyNumLastSlt.diValue			:= 0;
				tyP0400ProdSel.tyRcpDet.tyNumPitch.diValue				:= 0;
				tyP0400ProdSel.tyRcpDet.tyNumBrdPerSlt.diValue			:= 0;
				tyP0400ProdSel.tyRcpDet.tyBtnToptoBtm.bValue			:= FALSE;
				tyP0400ProdSel.tyRcpDet.tyBtnGapBetBrd.bValue			:= FALSE;
				tyP0400ProdSel.tyRcpDet.tyBtnLongBrd.bValue				:= FALSE;
				tyP0400ProdSel.tyRcpDet.tyNumMinReqFreeBffr.diValue		:= 0;
				tyP0400ProdSel.tyRcpDet.tyNumMtrPshrExtSpd.diValue		:= 0;
				tyP0400ProdSel.tyRcpDet.tyNumMtrPshrExtTorq.diValue		:= 0;
				tyP0400ProdSel.tyRcpDet.tyNumPshrOffset.diValue			:= p_tyProdRcpInfoOut.diPshrOffset;
			ELSE
				tyP0400ProdSel.tyRcpDet.tyStringRecipeNm.sValue			:= p_tyProdRcpInfoOut.sRcpNm;
				tyP0400ProdSel.tyRcpDet.tyNumProdWidth.diValue			:= p_tyProdRcpInfoOut.diWidthInUM;
				tyP0400ProdSel.tyRcpDet.tyNumProdWidth2.diValue			:= p_tyProdRcpInfoOut.diWidthInUM2;
				tyP0400ProdSel.tyRcpDet.tyTxtMcMode.usiValueIdx			:= p_tyProdRcpInfoOut.usiMcMod;
				tyP0400ProdSel.tyRcpDet.tyNumFirstSlt.diValue			:= p_tyProdRcpInfoOut.diMinSltValue;
				tyP0400ProdSel.tyRcpDet.tyNumLastSlt.diValue			:= p_tyProdRcpInfoOut.diMaxSltValue;
				tyP0400ProdSel.tyRcpDet.tyNumPitch.diValue				:= p_tyProdRcpInfoOut.diPitch;
				tyP0400ProdSel.tyRcpDet.tyNumBrdPerSlt.diValue			:= p_tyProdRcpInfoOut.diBrdPerSlt;
				tyP0400ProdSel.tyRcpDet.tyBtnToptoBtm.bValue			:= p_tyProdRcpInfoOut.bTopToBtm;
				tyP0400ProdSel.tyRcpDet.tyBtnGapBetBrd.bValue			:= p_tyProdRcpInfoOut.bGapBwtnBrd;
				tyP0400ProdSel.tyRcpDet.tyBtnLongBrd.bValue				:= p_tyProdRcpInfoOut.bLongBrd;
				tyP0400ProdSel.tyRcpDet.tyNumMinReqFreeBffr.diValue		:= p_tyProdRcpInfoOut.diMinReqFreeBffr;
				tyP0400ProdSel.tyRcpDet.tyNumMtrPshrExtSpd.diValue		:= p_tyProdRcpInfoOut.diMtrPshrExtSpd;
				tyP0400ProdSel.tyRcpDet.tyNumMtrPshrExtTorq.diValue		:= p_tyProdRcpInfoOut.diMtrPshrExtTorq;
				tyP0400ProdSel.tyRcpDet.tyNumPshrOffset.diValue			:= p_tyProdRcpInfoOut.diPshrOffset;
			END_IF

			fUIInRtStatOff(ADR(tyP0400ProdSel.tyRcpDet.tyLyr.uiRtStat));
			tyP0400ProdSel.tyProdSel.tyBtnPreview.bRtCompl	:= FALSE;

		END_IF

	END_IF

	IF tyP0400ProdSel.tyRcpDet.tyHotspotClose.bRtCompl = TRUE THEN
		tyP0400ProdSel.tyRcpDet.tyHotspotClose.bRtCompl	:= FALSE;
		tyP0400ProdSel.tyProdSel.tyBtnPreview.bValue	:= FALSE;

		//Hide Recipe Details
		fUIInRtStatHide(ADR(tyP0400ProdSel.tyRcpDet.tyLyr.uiRtStat));
	END_IF

	//254 Characters are Shown
	IF tyP0400ProdSel.tyRcpDet.tyHotspotShowLRcp.bRtCompl = TRUE THEN
		tyP0400ProdSel.tyRcpDet.tyHotspotShowLRcp.bRtCompl  := FALSE;

		fUIInRtStatOff(ADR(tyP0400ProdSel.tyRcpPopUp.tyLyr.uiRtStat));

		tyP0400ProdSel.tyRcpPopUp.tyStringInfo.sValue  :=  tyP0400ProdSel.tyProdSel.tyTableRecipe.a_tyStringDataCol1[tyP0400Table.uiSelectedRow].sValue; // Show 254 Characters

	ELSIF tyP0400ProdSel.tyRcpPopUp.tyHotspotClose.bRtCompl = TRUE THEN
		tyP0400ProdSel.tyRcpPopUp.tyHotspotClose.bRtCompl := FALSE;

		fUIInRtStatHide(ADR(tyP0400ProdSel.tyRcpPopUp.tyLyr.uiRtStat)); // Hide Pop Up Again

	END_IF

END_ACTION
```

#### Act_OptP0400Table.st
```iecst
ACTION Act_OptP0400Table:

	//Call Table FB
	fbP0400Table.sVisuNm			:= tyP0400Table.sVisuNm;
	fbP0400Table.udiWorkAreaStartX	:= 349;
	fbP0400Table.udiWorkAreaEndX	:= 768;
	fbP0400Table.udiWorkAreaStartY	:= 107;
	fbP0400Table.udiWorkAreaEndY	:= 428;
	fbP0400Table.udiMinXDist		:= 20;
	fbP0400Table.udiMinYDist		:= 20;
	fbP0400Table.uiSlideScale		:= c_uiP0400TableSize;
	fbP0400Table.iTotalData			:= UDINT_TO_INT(c_udiProdRcpMax);;
	fbP0400Table.iTotalRow			:= c_uiP0400TableSize;
	fbP0400Table(uiSliderStatus := tyP0400ProdSel.tyProdSel.tyTableRecipe.tyUISlider.uiRtStat , a_tyUIHotspot := tyP0400ProdSel.tyProdSel.tyTableRecipe.a_tyHotspot , uiTablePos := tyP0400Table.uiTablePos , iSliderPos := tyP0400ProdSel.tyProdSel.tyTableRecipe.tyUISlider.iValue);

	tyP0400Table.uiSelectedRow		:= fbP0400Table.uiSelectedRow;
	tyP0400Table.bTableActive		:= fbP0400Table.bTableActive;
	tyP0400Table.bSliderActive		:= fbP0400Table.bSliderActive;

	//Table Content
	iSelectedRowValue := STRING_TO_UINT(tyP0400ProdSel.tyProdSel.tyTableRecipe.a_tyStringDataCol0[tyP0400Table.uiSelectedRow].sValue);

	IF tyP0400Table.bTableActive = TRUE OR tyP0400Table.bSliderActive = TRUE OR bUpdateP0400Table THEN
		FOR i := 1 TO c_uiP0400TableSize DO
			IF tyP0400ProdSel.tyProdSel.tyBtnSort.bValue THEN

				tyP0400ProdSel.tyProdSel.tyTableRecipe.a_tyStringDataCol0[i].sValue	:= UINT_TO_STRING(tyP0400Table.uiTablePos + i - 1);
				tyP0400ProdSel.tyProdSel.tyTableRecipe.a_tyStringDataCol1[i].sValue	:= p_tyProdRcpSortedList[tyP0400Table.uiTablePos + i - 1].sRcpNm;
				tyP0400ProdSel.tyProdSel.tyTableRecipe.a_tyStringDataCol2[i].sValue	:= p_tyProdRcpSortedList[tyP0400Table.uiTablePos + i - 1].sDisplayInfo;

			ELSE

				IF tyP0400ProdSel.tyProdSel.tyStringSearch.sValue = '' THEN
					tyP0400ProdSel.tyProdSel.tyTableRecipe.a_tyStringDataCol0[i].sValue	:= UINT_TO_STRING(tyP0400Table.uiTablePos + i - 1);
					tyP0400ProdSel.tyProdSel.tyTableRecipe.a_tyStringDataCol1[i].sValue	:= p_tyProdRcpCurrList[tyP0400Table.uiTablePos + i - 1].sRcpNm;
					tyP0400ProdSel.tyProdSel.tyTableRecipe.a_tyStringDataCol2[i].sValue	:= p_tyProdRcpCurrList[tyP0400Table.uiTablePos + i - 1].sDisplayInfo;
				ELSE
					tyP0400ProdSel.tyProdSel.tyTableRecipe.a_tyStringDataCol0[i].sValue	:= UINT_TO_STRING(tyP0400Table.uiTablePos + i - 1);
					tyP0400ProdSel.tyProdSel.tyTableRecipe.a_tyStringDataCol1[i].sValue	:= p_tyProdRcpFilterList[tyP0400Table.uiTablePos + i - 1].sRcpNm;
					tyP0400ProdSel.tyProdSel.tyTableRecipe.a_tyStringDataCol2[i].sValue	:= p_tyProdRcpFilterList[tyP0400Table.uiTablePos + i - 1].sDisplayInfo;
				END_IF

			END_IF

		END_FOR

		IF bUpdateP0400Table THEN
			bUpdateP0400Table := FALSE;
		END_IF

	END_IF

	//Selected Row
	IF tyP0400Table.uiSelectedRow <> tyP0400Table.uiSelectedRowOld THEN
		FOR i := 1 TO c_uiP0400TableSize DO
			IF tyP0400Table.uiSelectedRow = i THEN
				tyP0400ProdSel.tyProdSel.tyTableRecipe.a_tyStringDataCol1[i].usiColor	:= 1;
				tyP0400ProdSel.tyProdSel.tyTableRecipe.a_tyStringDataCol2[i].usiColor	:= 1;
			ELSE
				tyP0400ProdSel.tyProdSel.tyTableRecipe.a_tyStringDataCol1[i].usiColor	:= 0;
				tyP0400ProdSel.tyProdSel.tyTableRecipe.a_tyStringDataCol2[i].usiColor	:= 0;
			END_IF
		END_FOR

		tyP0400Table.uiSelectedRowOld	:= tyP0400Table.uiSelectedRow;
	END_IF

END_ACTION
```

#### Act_OptP0400Keypad.st
```iecst
ACTION Act_OptP0400Keypad:

	IF fUIOutRtStatTPIsOpen(ADR(tyP0400ProdSel.tyProdSel.tyStringSearch.uiRtStat)) THEN
		tyProperty.tyKeypad.tyStringTitle.sKeypadTitle	:= tyP0400ProdSel.tyProdSel.tyStringSearch.sKeypadTitle;

	ELSE
		tyProperty.tyKeypad.tyStringTitle.sKeypadTitle	:= '';

	END_IF

END_ACTION
```

#### Act_EntP0410Disp.st
```iecst
ACTION Act_EntP0410Disp:

	//Access Addres
	p_tyC0005Main ACCESS ADR(tyCommon.tyMain);

	p_tyC0007Notif ACCESS ADR(tyCommon.tyNotif);

	p_tyC0008MsgBox ACCESS ADR(tyP0410MagSel.tyMsgBoxHide);

	p_tyC0009Info ACCESS ADR(tyCommon.tyInfo);

	p_tyP0410MagSel ACCESS ADR(tyP0410MagSel.tyMagSel);
	p_tyP0410MagDet ACCESS ADR(tyP0410MagSel.tyMagDet);

	tyP0410MagSel.tyMagSel.tyBtnSort.bValue 	:= FALSE;
	tyP0410MagSel.tyMagSel.tyBtnSort.bRtCompl 	:= FALSE;

	bRefreshMagRcpTable := TRUE;

	fUIInRtStatHide(ADR(tyP0410MagSel.tyMagDet.tyLyr.uiRtStat));

	// Enabling Display Auto Detect Magazine Mode
	tyP0410MagSel.tyMagSel.tyTxtMagModel.uiRtStat :=  NOT(p_tyNtParamCurr.bMagAutoVerifyPrep);

END_ACTION
```

#### Act_OptP0410Mask.st
```iecst
ACTION Act_OptP0410Mask:

	IF tyP0410MagSel.tyMagSel.tyBtnLoad.bRtCompl = FALSE THEN
		IF tyP0410MagSel.tyMagSel.tyTableRecipe.a_tyStringDataCol1[tyP0410Table.uiSelectedRow].sValue = '' THEN
			fUIInRtStatOff(ADR(tyP0410MagSel.tyMagSel.tyBtnLoad.uiMaskRtStat));
			fUIInRtStatOff(ADR(tyP0410MagSel.tyMagSel.tyBtnPreview.uiMaskRtStat));
		ELSE
			fUIInRtStatHide(ADR(tyP0410MagSel.tyMagSel.tyBtnLoad.uiMaskRtStat));
			fUIInRtStatHide(ADR(tyP0410MagSel.tyMagSel.tyBtnPreview.uiMaskRtStat));
		END_IF
	END_IF

	tyP0410MagSel.tyMagSel.tyBtnSort.uiMaskRtStat.0		:= (tyP0410MagSel.tyMagSel.tyTableRecipe.a_tyStringDataCol1[1].sValue <> '') AND (tyP0410MagSel.tyMagSel.tyBtnLoad.bRtCompl = FALSE);

END_ACTION
```

#### Act_OptP0410Load.st
```iecst
ACTION Act_OptP0410Load:

	IF tyP0410MagSel.tyMagSel.tyBtnLoad.bRtCompl = TRUE THEN

		IF usiSelMagRcpStep = 0 THEN
			//Message Confirmation Ask
			//Mask
			tyP0410MagSel.tyMagSel.tyTableRecipe.uiMaskRtStat.0		:= FALSE;
			tyP0410MagSel.tyMagSel.tyBtnPreview.uiMaskRtStat.0		:= FALSE;

			p_tyC0008MsgBox ACCESS ADR(tyP0410MagSel.tyMsgBoxSelRcpAsk);

			IF tyP0410MagSel.tyMsgBoxSelRcpAsk.tyBtnYes.bRtCompl = TRUE THEN
				tyP0410MagSel.tyMsgBoxSelRcpAsk.tyBtnYes.bRtCompl	:= FALSE;
				tyP0410MagSel.tyMsgBoxSelRcpAsk.tyBtnYes.bValue		:= FALSE;

				p_tyC0008MsgBox ACCESS ADR(tyP0410MagSel.tyMsgBoxHide);

				usiSelMagRcpStep		:= 1;

			ELSIF tyP0410MagSel.tyMsgBoxSelRcpAsk.tyBtnNo.bRtCompl = TRUE THEN
				tyP0410MagSel.tyMsgBoxSelRcpAsk.tyBtnNo.bRtCompl	:= FALSE;
				tyP0410MagSel.tyMsgBoxSelRcpAsk.tyBtnNo.bValue		:= FALSE;

				p_tyC0008MsgBox ACCESS ADR(tyP0410MagSel.tyMsgBoxHide);

				usiSelMagRcpStep		:= 99;

			END_IF

		ELSIF usiSelMagRcpStep = 1 THEN
			//Load Magazine Recipe
			tyMagRcpInfoIn.sRcpNm		:= tyP0410MagSel.tyMagSel.tyTableRecipe.a_tyStringDataCol1[tyP0410Table.uiSelectedRow].sValue;

			eMagRcpAct	:= MagRcpActLoadRcp;

			IF p_eMagRcpStat = MagRcpActLoadRcp AND p_eMagRcpStatus = Done THEN
				eMagRcpAct	:= MagRcpActIdle;

				IF p_bMagRcpNmEmpty = TRUE AND p_bMagRcpNmNotExist = TRUE THEN
					usiSelMagRcpStep	:= 2;
				ELSE
					//Update UI Current Recipe
					tyP0410MagSel.tyMagSel.tyStringRecipeNm.sValue			:= p_tyMagRcpCurrRcp.sRcpNm;
					tyP0410MagSel.tyMagSel.tyNumSltToSltDist.diValue		:= p_tyMagRcpCurrRcp.diSltToSltInUM;
					tyP0410MagSel.tyMagSel.tyNumMaxSlt.diValue				:= p_tyMagRcpCurrRcp.diTtlSlt;
					tyP0410MagSel.tyMagSel.tyNumLifterMag1Slt1Pos.diValue	:= p_tyMagRcpCurrRcp.diMag1Slt1PosInUM;
					tyP0410MagSel.tyMagSel.tyNumLifterMag2Slt1Pos.diValue	:= p_tyMagRcpCurrRcp.diMag2Slt1PosInUM;
					tyP0410MagSel.tyMagSel.tyNumLifterMag3Slt1Pos.diValue	:= p_tyMagRcpCurrRcp.diMag3Slt1PosInUM;
					tyP0410MagSel.tyMagSel.tyNumTravPosMag1.diValue			:= p_tyMagRcpCurrRcp.diMag1TravPosInUM;
					tyP0410MagSel.tyMagSel.tyNumTravPosMag2.diValue			:= p_tyMagRcpCurrRcp.diMag2TravPosInUM;
					tyP0410MagSel.tyMagSel.tyNumTravPosMag3.diValue			:= p_tyMagRcpCurrRcp.diMag3TravPosInUM;
					tyP0410MagSel.tyMagSel.tyTxtMagModel.usiValueIdx		:= p_tyMagRcpCurrRcp.usiMagModel;
					tyP0410MagSel.tyMagSel.tyNumMagMaxBrdWidth.diValue		:= p_tyMagRcpCurrRcp.diMagMaxBrdWidth;
					tyP0410MagSel.tyMagSel.tyBtnSafetyBar.bValue			:= p_tyMagRcpCurrRcp.bSafetyBarDisabled;
					tyP0410MagSel.tyMagSel.tyBtnMagHeightChkEn.bValue		:= p_tyMagRcpCurrRcp.bMagHeightChkEn;

					tyMagRcpCurrRcpWr	:= p_tyMagRcpCurrRcp;

					usiSelMagRcpStep	:= 99;
				END_IF

			ELSIF p_eProdRcpStatus = Error THEN

				usiSelMagRcpStep		:= 99;

			END_IF

		ELSIF usiSelMagRcpStep = 2 THEN
			//Message Name Not Found
			p_tyC0008MsgBox ACCESS ADR(tyP0410MagSel.tyMsgBoxSelRcpNoNm);

			IF tyP0410MagSel.tyMsgBoxSelRcpNoNm.tyBtnNo.bRtCompl = TRUE THEN
				tyP0410MagSel.tyMsgBoxSelRcpNoNm.tyBtnNo.bRtCompl	:= FALSE;
				tyP0410MagSel.tyMsgBoxSelRcpNoNm.tyBtnNo.bValue		:= FALSE;

				p_tyC0008MsgBox ACCESS ADR(tyP0410MagSel.tyMsgBoxHide);

				usiSelMagRcpStep		:= 99;

			END_IF

		ELSIF usiSelMagRcpStep = 99 THEN
			//Complete
			//Unmask
			tyP0410MagSel.tyMagSel.tyTableRecipe.uiMaskRtStat.0		:= TRUE;
			tyP0410MagSel.tyMagSel.tyBtnPreview.uiMaskRtStat.0		:= TRUE;

			//Reset
			tyP0410MagSel.tyMagSel.tyBtnLoad.bRtCompl				:= FALSE;
			tyP0410MagSel.tyMagSel.tyBtnLoad.bValue					:= FALSE;

			usiSelMagRcpStep			:= 0;

		END_IF

	END_IF

END_ACTION
```

#### Act_OptP0410Preview.st
```iecst
ACTION Act_OptP0410Preview:

	IF tyP0410MagSel.tyMagSel.tyBtnPreview.bRtCompl = TRUE THEN

		tyMagRcpInfoIn.sRcpNm	:= tyP0410MagSel.tyMagSel.tyTableRecipe.a_tyStringDataCol1[tyP0410Table.uiSelectedRow].sValue;

		eMagRcpAct				:= MagRcpActGetInfo;

		IF	p_eMagRcpStat = MagRcpActGetInfo AND p_eMagRcpStatus = Done THEN
			eMagRcpAct			:= MagRcpActIdle;

			IF p_bMagRcpNmEmpty = TRUE AND p_bMagRcpNmNotExist = TRUE THEN

				tyP0410MagSel.tyMagDet.tyStringRecipeNm.sValue			:= '';
				tyP0410MagSel.tyMagDet.tyNumSltToSltDist.diValue		:= 0;
				tyP0410MagSel.tyMagDet.tyNumMaxSlt.diValue				:= 0;
				tyP0410MagSel.tyMagDet.tyNumLifterMag1Slt1Pos.diValue	:= 0;
				tyP0410MagSel.tyMagDet.tyNumLifterMag2Slt1Pos.diValue	:= 0;
				tyP0410MagSel.tyMagDet.tyNumLifterMag3Slt1Pos.diValue	:= 0;
				tyP0410MagSel.tyMagDet.tyNumTravPosMag1.diValue			:= 0;
				tyP0410MagSel.tyMagDet.tyNumTravPosMag2.diValue			:= 0;
				tyP0410MagSel.tyMagDet.tyNumTravPosMag3.diValue			:= 0;
				tyP0410MagSel.tyMagDet.tyNumMagMaxBrdWidth.diValue		:= 0;
				tyP0410MagSel.tyMagDet.tyBtnSafetyBar.bValue			:= FALSE;
				tyP0410MagSel.tyMagDet.tyBtnMagHeightChkEn.bValue		:= FALSE;
			ELSE

				tyP0410MagSel.tyMagDet.tyStringRecipeNm.sValue			:= p_tyMagRcpInfoOut.sRcpNm;
				tyP0410MagSel.tyMagDet.tyNumSltToSltDist.diValue		:= p_tyMagRcpInfoOut.diSltToSltInUM;
				tyP0410MagSel.tyMagDet.tyNumMaxSlt.diValue				:= p_tyMagRcpInfoOut.diTtlSlt;
				tyP0410MagSel.tyMagDet.tyNumLifterMag1Slt1Pos.diValue	:= p_tyMagRcpInfoOut.diMag1Slt1PosInUM;
				tyP0410MagSel.tyMagDet.tyNumLifterMag2Slt1Pos.diValue	:= p_tyMagRcpInfoOut.diMag2Slt1PosInUM;
				tyP0410MagSel.tyMagDet.tyNumLifterMag3Slt1Pos.diValue	:= p_tyMagRcpInfoOut.diMag3Slt1PosInUM;
				tyP0410MagSel.tyMagDet.tyNumTravPosMag1.diValue			:= p_tyMagRcpInfoOut.diMag1TravPosInUM;
				tyP0410MagSel.tyMagDet.tyNumTravPosMag2.diValue			:= p_tyMagRcpInfoOut.diMag2TravPosInUM;
				tyP0410MagSel.tyMagDet.tyNumTravPosMag3.diValue			:= p_tyMagRcpInfoOut.diMag3TravPosInUM;
				tyP0410MagSel.tyMagDet.tyNumMagMaxBrdWidth.diValue		:= p_tyMagRcpInfoOut.diMagMaxBrdWidth;
				tyP0410MagSel.tyMagDet.tyBtnSafetyBar.bValue			:= p_tyMagRcpInfoOut.bSafetyBarDisabled;
				tyP0410MagSel.tyMagDet.tyBtnMagHeightChkEn.bValue		:= p_tyMagRcpInfoOut.bMagHeightChkEn;
			END_IF

			fUIInRtStatOff(ADR(tyP0410MagSel.tyMagDet.tyLyr.uiRtStat));

			tyP0410MagSel.tyMagSel.tyBtnPreview.bRtCompl				:= FALSE;
		END_IF

	END_IF

	IF tyP0410MagSel.tyMagDet.tyHotspotClose.bRtCompl = TRUE THEN
		tyP0410MagSel.tyMagDet.tyHotspotClose.bRtCompl					:= FALSE;
		tyP0410MagSel.tyMagSel.tyBtnPreview.bValue						:= FALSE;

		//Hide Recipe Details
		fUIInRtStatHide(ADR(tyP0410MagSel.tyMagDet.tyLyr.uiRtStat));
	END_IF

END_ACTION
```

#### Act_OptP0410Table.st
```iecst
ACTION Act_OptP0410Table:

	//Call Table FB
	fbP0410Table.sVisuNm			:= tyP0410Table.sVisuNm;
	fbP0410Table.udiWorkAreaStartX	:= 349;
	fbP0410Table.udiWorkAreaEndX	:= 768;
	fbP0410Table.udiWorkAreaStartY	:= 107;
	fbP0410Table.udiWorkAreaEndY	:= 428;
	fbP0410Table.udiMinXDist		:= 20;
	fbP0410Table.udiMinYDist		:= 20;
	fbP0410Table.uiSlideScale		:= c_uiP0410TableSize;
	fbP0410Table.iTotalData			:= UDINT_TO_INT(c_udiMagRcpMax);;
	fbP0410Table.iTotalRow			:= c_uiP0410TableSize;
	fbP0410Table(uiSliderStatus := tyP0410MagSel.tyMagSel.tyTableRecipe.tyUISlider.uiRtStat , a_tyUIHotspot := tyP0410MagSel.tyMagSel.tyTableRecipe.a_tyHotspot , uiTablePos := tyP0410Table.uiTablePos , iSliderPos := tyP0410MagSel.tyMagSel.tyTableRecipe.tyUISlider.iValue);

	tyP0410Table.uiSelectedRow		:= fbP0410Table.uiSelectedRow;
	tyP0410Table.bTableActive		:= fbP0410Table.bTableActive;
	tyP0410Table.bSliderActive		:= fbP0410Table.bSliderActive;

	//Table Content
	IF tyP0410Table.bTableActive = TRUE OR tyP0410Table.bSliderActive = TRUE OR bRefreshMagRcpTable OR bUpdateP0410Table THEN
		FOR i := 1 TO c_uiP0410TableSize DO
			IF tyP0410MagSel.tyMagSel.tyBtnSort.bValue THEN

				tyP0410MagSel.tyMagSel.tyTableRecipe.a_tyStringDataCol0[i].sValue	:= UINT_TO_STRING(tyP0410Table.uiTablePos + i - 1);
				tyP0410MagSel.tyMagSel.tyTableRecipe.a_tyStringDataCol1[i].sValue	:= p_tyMagRcpSortedList[tyP0410Table.uiTablePos + i - 1].sRcpNm;
				tyP0410MagSel.tyMagSel.tyTableRecipe.a_tyStringDataCol2[i].sValue	:= p_tyMagRcpSortedList[tyP0410Table.uiTablePos + i - 1].sDisplayInfo;

			ELSE
				tyP0410MagSel.tyMagSel.tyTableRecipe.a_tyStringDataCol0[i].sValue	    := UINT_TO_STRING(tyP0410Table.uiTablePos + i - 1);
				tyP0410MagSel.tyMagSel.tyTableRecipe.a_tyStringDataCol1[i].sValue		:= p_tyMagRcpCurrList[tyP0410Table.uiTablePos + i - 1].sRcpNm;
				tyP0410MagSel.tyMagSel.tyTableRecipe.a_tyStringDataCol2[i].sValue		:= p_tyMagRcpCurrList[tyP0410Table.uiTablePos + i - 1].sDisplayInfo;
			END_IF

		END_FOR

		IF bUpdateP0410Table THEN
			bUpdateP0410Table := FALSE;
		END_IF
	END_IF

	//Selected Row
	IF tyP0410Table.uiSelectedRow <> tyP0410Table.uiSelectedRowOld THEN
		FOR i := 1 TO c_uiP0410TableSize DO
			IF tyP0410Table.uiSelectedRow = i THEN
				tyP0410MagSel.tyMagSel.tyTableRecipe.a_tyStringDataCol1[i].usiColor	:= 1;
				tyP0410MagSel.tyMagSel.tyTableRecipe.a_tyStringDataCol2[i].usiColor	:= 1;
			ELSE
				tyP0410MagSel.tyMagSel.tyTableRecipe.a_tyStringDataCol1[i].usiColor	:= 0;
				tyP0410MagSel.tyMagSel.tyTableRecipe.a_tyStringDataCol2[i].usiColor	:= 0;
			END_IF
		END_FOR

		tyP0410Table.uiSelectedRowOld	:= tyP0410Table.uiSelectedRow;
	END_IF

END_ACTION
```

#### Act_OptP0410Sort.st
```iecst
ACTION Act_OptP0410Sort:

	IF tyP0410MagSel.tyMagSel.tyBtnSort.bValue THEN
		tyP0410MagSel.tyMagSel.tyBtnSort.usiTxtIdx 	:= 1;
	ELSE
		tyP0410MagSel.tyMagSel.tyBtnSort.usiTxtIdx 	:= 0;
	END_IF

	IF tyP0410MagSel.tyMagSel.tyBtnSort.bRtCompl THEN

		IF tyP0410MagSel.tyMagSel.tyBtnSort.bValue THEN

			tyP0410MagSel.tyMagSel.tyTableRecipe.uiMaskRtStat.0	:= FALSE;

			eMagRcpAct	:= MagRcpActSort;

			IF p_eMagRcpStat = MagRcpActSort AND p_eMagRcpStatus = Done THEN
				eMagRcpAct		:= MagRcpActIdle;

				FOR i := 1 TO c_uiP0410TableSize DO
					tyP0410MagSel.tyMagSel.tyTableRecipe.a_tyStringDataCol0[i].sValue	:= UINT_TO_STRING(tyP0400Table.uiTablePos + i - 1);
					tyP0410MagSel.tyMagSel.tyTableRecipe.a_tyStringDataCol1[i].sValue	:= p_tyMagRcpSortedList[tyP0400Table.uiTablePos + i - 1].sRcpNm;
					tyP0410MagSel.tyMagSel.tyTableRecipe.a_tyStringDataCol2[i].sValue	:= p_tyMagRcpSortedList[tyP0400Table.uiTablePos + i - 1].sDisplayInfo;
				END_FOR

				//Unmask
				tyP0410MagSel.tyMagSel.tyTableRecipe.uiMaskRtStat.0	:= TRUE;

				tyP0410MagSel.tyMagSel.tyBtnSort.bRtCompl := FALSE;

			ELSIF p_eMagRcpStatus = Error THEN
				FOR i := 1 TO c_uiP0410TableSize DO
					tyP0410MagSel.tyMagSel.tyTableRecipe.a_tyStringDataCol0[i].sValue		:= UINT_TO_STRING(tyP0410Table.uiTablePos + i - 1);
					tyP0410MagSel.tyMagSel.tyTableRecipe.a_tyStringDataCol1[i].sValue		:= '';
					tyP0410MagSel.tyMagSel.tyTableRecipe.a_tyStringDataCol2[i].sValue		:= '';
				END_FOR

				p_tyC0008MsgBox ACCESS ADR (tyP0410MagSel.tyMsgBoxListErr);

				IF tyP0410MagSel.tyMsgBoxListErr.tyBtnNo.bRtCompl = TRUE THEN
					tyP0410MagSel.tyMsgBoxListErr.tyBtnNo.bRtCompl 		:= TRUE;
					tyP0410MagSel.tyMsgBoxListErr.tyBtnNo.bValue			:= TRUE;

					p_tyC0008MsgBox ACCESS ADR (tyP0410MagSel.tyMsgBoxHide);

					//Unmask
					tyP0410MagSel.tyMagSel.tyTableRecipe.uiMaskRtStat.0	:= TRUE;

					//Reset
					tyP0410MagSel.tyMagSel.tyBtnSort.bRtCompl := FALSE;
				END_IF
			END_IF

		ELSE

			bUpdateP0410Table	:= TRUE;

			tyP0410MagSel.tyMagSel.tyBtnSort.bRtCompl := FALSE;

		END_IF

	END_IF

END_ACTION
```

#### Act_EntP0600Disp.st
```iecst
ACTION Act_EntP0600Disp:

	//Access Addres
	p_tyC0005Main ACCESS ADR(tyCommon.tyMain);

	p_tyC0007Notif ACCESS ADR(tyCommon.tyNotif);

	p_tyC0008MsgBox ACCESS ADR(tyP0600Alm.tyMsgBoxHide);

	p_tyC0009Info ACCESS ADR(tyCommon.tyInfo);

	p_tyC0010RcyMsg ACCESS ADR(tyP0600Alm.tyRcyMsgHide);

	p_tyP0600Alm ACCESS ADR(tyP0600Alm.tyAlm);

	tyP0600Alm.tyAlm.tyBtnCurr.bRtCompl := TRUE; //Default will be Current Alarm View

	//Reset
	bTeachTravPosA			:= FALSE;
	bTeachTravPosB			:= FALSE;
	bTeachLifterPosA		:= FALSE;
	bTeachLifterPosB		:= FALSE;
	bTeachLifterMag1Slt1Pos	:= FALSE;
	bTeachLifterMag2Slt1Pos	:= FALSE;
	bTeachLifterMag3Slt1Pos	:= FALSE;
	bTeachTravPosMag1		:= FALSE;
	bTeachTravPosMag2		:= FALSE;
	bTeachTravPosMag3		:= FALSE;
	bTeachLifterTopPos	:= FALSE;
	bTeachLifterBtmPos	:= FALSE;
	bTeachLifterTopPos2	:= FALSE;
	bTeachLifterBtmPos2	:= FALSE;

END_ACTION
```

#### Act_OptP0600RcyMsg.st
```iecst
ACTION Act_OptP0600RcyMsg:

	//Recovery Message
	FOR i := 1 TO c_uiP0600TableSize DO

		IF tyP0600Alm.tyAlm.a_tyHotspotAlm[i].bRtCompl = TRUE THEN
			tyP0600Alm.tyAlm.a_tyHotspotAlm[i].bRtCompl	:= FALSE;

			tyP0600Alm.tyRcyMsg.tyTxtMsg.udiValueIdx := p_tyAlarmRcyList[i];

			IF tyP0600Alm.tyRcyMsg.tyTxtMsg.udiValueIdx <> 0 AND tyP0600Alm.tyAlm.tyBtnHistory.bValue = FALSE THEN
				p_tyC0010RcyMsg ACCESS ADR(tyP0600Alm.tyRcyMsg);
			ELSE
				p_tyC0010RcyMsg ACCESS ADR(tyP0600Alm.tyRcyMsgHide);
			END_IF

		END_IF

	END_FOR

	// Close Recovery Message
	IF tyP0600Alm.tyRcyMsg.tyHotspotClose.bRtCompl THEN
		tyP0600Alm.tyRcyMsg.tyHotspotClose.bRtCompl := FALSE;

		p_tyC0010RcyMsg ACCESS ADR(tyP0600Alm.tyRcyMsgHide);
	END_IF

END_ACTION
```

#### Act_OptP0600Alm.st
```iecst
ACTION Act_OptP0600Alm:

	IF tyP0600Alm.tyAlm.tyBtnHistory.bRtCompl = TRUE THEN
		tyP0600Alm.tyAlm.tyBtnHistory.bRtCompl		:= FALSE;
		tyP0600Alm.tyAlm.tyBtnHistory.bValue		:= TRUE;
		tyP0600Alm.tyAlm.tyBtnCurr.bValue			:= FALSE;
	ELSIF tyP0600Alm.tyAlm.tyBtnCurr.bRtCompl = TRUE THEN
		tyP0600Alm.tyAlm.tyBtnCurr.bRtCompl			:= FALSE;
		tyP0600Alm.tyAlm.tyBtnCurr.bValue			:= TRUE;
		tyP0600Alm.tyAlm.tyBtnHistory.bValue		:= FALSE;
	END_IF

	IF NOT p_bAlarmErr THEN
		memset(ADR(tyUIAlmData.bAlm) , 0 , SIZEOF(tyUIAlmData.bAlm));
	END_IF

	IF NOT p_bAlarmWarning THEN
		memset(ADR(tyUIAlmData.bWarning) , 0 , SIZEOF(tyUIAlmData.bWarning));
	ELSE
		IF p_bUSHermesAConnected OR p_tyMcParamCurr.eUSCommA = McSetCommModSMEMA THEN
			tyUIAlmData.bWarning[3114] := FALSE;
		END_IF
		IF p_bUSHermesBConnected OR p_tyMcParamCurr.eUSCommB = McSetCommModSMEMA THEN
			tyUIAlmData.bWarning[3281] := FALSE;
		END_IF
	END_IF

	IF tyP0600Alm.tyAlm.tyBtnCurr.bValue = TRUE THEN

		fUIInRtStatOff(ADR(tyP0600Alm.tyAlm.tyAlarm.tyUIAlmCur.uiRtStat));
		fUIInRtStatHide(ADR(tyP0600Alm.tyAlm.tyAlarm.tyUIAlmHis.uiRtStat));
		tyP0600Alm.tyAlm.tyBtnHistoryUp.uiMaskRtStat.0 		:= FALSE;
		tyP0600Alm.tyAlm.tyBtnHistoryDown.uiMaskRtStat.0 	:= FALSE;

		FOR i := 1 TO c_uiP0600TableSize DO
			IF p_bStartupUISettingsLoadDone THEN
				IF p_tyAlarmCurrList[i].eSeverity = AlmSeverityError THEN
					tyUIAlmData.bAlm[p_tyAlarmCurrList[i].udiErrorCode] := p_tyAlarmCurrList[i].bAlm;
				ELSIF p_tyAlarmCurrList[i].eSeverity = AlmSeverityWarning THEN
					tyUIAlmData.bWarning[p_tyAlarmCurrList[i].udiErrorCode] := p_tyAlarmCurrList[i].bWarning;
				END_IF
			END_IF
		END_FOR

	ELSIF tyP0600Alm.tyAlm.tyBtnHistory.bValue = TRUE THEN

		fUIInRtStatHide(ADR(tyP0600Alm.tyAlm.tyAlarm.tyUIAlmCur.uiRtStat));
		fUIInRtStatOff(ADR(tyP0600Alm.tyAlm.tyAlarm.tyUIAlmHis.uiRtStat));
		tyP0600Alm.tyAlm.tyBtnHistoryUp.uiMaskRtStat.0 		:= TRUE;
		tyP0600Alm.tyAlm.tyBtnHistoryDown.uiMaskRtStat.0 	:= TRUE;

	END_IF

END_ACTION
```

#### Act_EntP0700Disp.st
```iecst
ACTION Act_EntP0700Disp:

	//Access Address
	p_tyC0005Main ACCESS ADR(tyCommon.tyMain);

	p_tyC0007Notif ACCESS ADR(tyCommon.tyNotif);

	p_tyC0008MsgBox ACCESS ADR(tyP0700LFCtrl.tyMsgBoxHide);

	p_tyC0009Info ACCESS ADR(tyCommon.tyInfo);

	p_tyP0700LFCtrl ACCESS ADR(tyP0700LFCtrl.tyLdr);

	//Run
	bLeaderRun	:= TRUE;

END_ACTION
```

#### Act_ExitP0700.st
```iecst
ACTION Act_ExitP0700:

	IF NOT(tyP0700LFCtrl.tyLdr.tyBtnChgAll.bRtCompl OR tyP0700LFCtrl.tyLdr.tyBtnChgSeqAuto.bRtCompl OR tyP0700LFCtrl.tyLdr.tyBtnChgSeqMnl.bRtCompl OR tyP0700LFCtrl.tyLdr.tyBtnSyncTm.bRtCompl) THEN
		bLeaderRun	:= FALSE;
		bLFRunInBG	:= FALSE;
	ELSE
		bLFRunInBG	:= TRUE;
	END_IF

	usiChgPage	:= 1;

END_ACTION
```

#### Act_OptP0700LFLeaderCtrl.st
```iecst
ACTION Act_OptP0700LFLeaderCtrl:

	CASE usiLFLeaderCtrlStep OF
		0:	//Confirmation Message - Execute Ask
			IF tyP0700LFCtrl.tyLdr.tyBtnChgAll.bRtCompl THEN

				p_tyC0008MsgBox ACCESS ADR(tyP0700LFCtrl.tyMsgBoxChgAllAsk);

				IF tyP0700LFCtrl.tyMsgBoxChgAllAsk.tyBtnYes.bRtCompl = TRUE THEN
					tyP0700LFCtrl.tyMsgBoxChgAllAsk.tyBtnYes.bRtCompl	:= FALSE;
					tyP0700LFCtrl.tyMsgBoxChgAllAsk.tyBtnYes.bValue		:= FALSE;

					p_tyC0008MsgBox ACCESS ADR(tyP0700LFCtrl.tyMsgBoxHide);

					tyP0700LFCtrl.tyLdr.tyBtnChgAll.bValue		:= TRUE;

					usiLFLeaderCtrlStep	:= 2;

				ELSIF tyP0700LFCtrl.tyMsgBoxChgAllAsk.tyBtnNo.bRtCompl = TRUE THEN
					tyP0700LFCtrl.tyMsgBoxChgAllAsk.tyBtnNo.bRtCompl	:= FALSE;
					tyP0700LFCtrl.tyMsgBoxChgAllAsk.tyBtnNo.bValue		:= FALSE;

					p_tyC0008MsgBox ACCESS ADR(tyP0700LFCtrl.tyMsgBoxHide);

					tyP0700LFCtrl.tyLdr.tyBtnChgAll.bValue		:= FALSE;
					tyP0700LFCtrl.tyLdr.tyBtnChgAll.bRtCompl	:= FALSE;

				END_IF

			ELSIF tyP0700LFCtrl.tyLdr.tyBtnChgSeqAuto.bRtCompl THEN

				p_tyC0008MsgBox ACCESS ADR(tyP0700LFCtrl.tyMsgBoxChgSeqAutoAsk);

				IF tyP0700LFCtrl.tyMsgBoxChgSeqAutoAsk.tyBtnYes.bRtCompl = TRUE THEN
					tyP0700LFCtrl.tyMsgBoxChgSeqAutoAsk.tyBtnYes.bRtCompl	:= FALSE;
					tyP0700LFCtrl.tyMsgBoxChgSeqAutoAsk.tyBtnYes.bValue		:= FALSE;

					p_tyC0008MsgBox ACCESS ADR(tyP0700LFCtrl.tyMsgBoxHide);

					tyP0700LFCtrl.tyLdr.tyBtnChgSeqAuto.bValue		:= TRUE;

					usiLFLeaderCtrlStep	:= 2;

				ELSIF tyP0700LFCtrl.tyMsgBoxChgSeqAutoAsk.tyBtnNo.bRtCompl = TRUE THEN
					tyP0700LFCtrl.tyMsgBoxChgSeqAutoAsk.tyBtnNo.bRtCompl	:= FALSE;
					tyP0700LFCtrl.tyMsgBoxChgSeqAutoAsk.tyBtnNo.bValue		:= FALSE;

					p_tyC0008MsgBox ACCESS ADR(tyP0700LFCtrl.tyMsgBoxHide);

					tyP0700LFCtrl.tyLdr.tyBtnChgSeqAuto.bValue		:= FALSE;
					tyP0700LFCtrl.tyLdr.tyBtnChgSeqAuto.bRtCompl	:= FALSE;

				END_IF

			ELSIF tyP0700LFCtrl.tyLdr.tyBtnChgSeqMnl.bRtCompl THEN

				p_tyC0008MsgBox ACCESS ADR(tyP0700LFCtrl.tyMsgBoxChgSeqMnlAsk);

				IF tyP0700LFCtrl.tyMsgBoxChgSeqMnlAsk.tyBtnYes.bRtCompl = TRUE THEN
					tyP0700LFCtrl.tyMsgBoxChgSeqMnlAsk.tyBtnYes.bRtCompl	:= FALSE;
					tyP0700LFCtrl.tyMsgBoxChgSeqMnlAsk.tyBtnYes.bValue		:= FALSE;

					p_tyC0008MsgBox ACCESS ADR(tyP0700LFCtrl.tyMsgBoxHide);

					tyP0700LFCtrl.tyLdr.tyBtnChgSeqMnl.bValue	:= TRUE;

					usiLFLeaderCtrlStep	:= 2;

				ELSIF tyP0700LFCtrl.tyMsgBoxChgSeqMnlAsk.tyBtnNo.bRtCompl = TRUE THEN
					tyP0700LFCtrl.tyMsgBoxChgSeqMnlAsk.tyBtnNo.bRtCompl		:= FALSE;
					tyP0700LFCtrl.tyMsgBoxChgSeqMnlAsk.tyBtnNo.bValue		:= FALSE;

					p_tyC0008MsgBox ACCESS ADR(tyP0700LFCtrl.tyMsgBoxHide);

					tyP0700LFCtrl.tyLdr.tyBtnChgSeqMnl.bValue	:= FALSE;
					tyP0700LFCtrl.tyLdr.tyBtnChgSeqMnl.bRtCompl	:= FALSE;

				END_IF

			ELSIF tyP0700LFCtrl.tyLdr.tyBtnSyncTm.bRtCompl THEN

				p_tyC0008MsgBox ACCESS ADR(tyP0700LFCtrl.tyMsgBoxSyncPLCTmAsk);

				IF tyP0700LFCtrl.tyMsgBoxSyncPLCTmAsk.tyBtnYes.bRtCompl = TRUE THEN
					tyP0700LFCtrl.tyMsgBoxSyncPLCTmAsk.tyBtnYes.bRtCompl	:= FALSE;
					tyP0700LFCtrl.tyMsgBoxSyncPLCTmAsk.tyBtnYes.bValue		:= FALSE;

					p_tyC0008MsgBox ACCESS ADR(tyP0700LFCtrl.tyMsgBoxHide);

					tyP0700LFCtrl.tyLdr.tyBtnSyncTm.bValue		:= TRUE;

					usiLFLeaderCtrlStep	:= 2;

				ELSIF tyP0700LFCtrl.tyMsgBoxSyncPLCTmAsk.tyBtnNo.bRtCompl = TRUE THEN
					tyP0700LFCtrl.tyMsgBoxSyncPLCTmAsk.tyBtnNo.bRtCompl		:= FALSE;
					tyP0700LFCtrl.tyMsgBoxSyncPLCTmAsk.tyBtnNo.bValue		:= FALSE;

					p_tyC0008MsgBox ACCESS ADR(tyP0700LFCtrl.tyMsgBoxHide);

					tyP0700LFCtrl.tyLdr.tyBtnSyncTm.bValue		:= FALSE;
					tyP0700LFCtrl.tyLdr.tyBtnSyncTm.bRtCompl	:= FALSE;

				END_IF

			END_IF

		1:	//Confirmation Message - Terminate Ask
			p_tyC0008MsgBox ACCESS ADR(tyP0700LFCtrl.tyMsgBoxTerminateOpsAsk);

			IF tyP0700LFCtrl.tyMsgBoxTerminateOpsAsk.tyBtnYes.bRtCompl = TRUE THEN
				tyP0700LFCtrl.tyMsgBoxTerminateOpsAsk.tyBtnYes.bRtCompl	:= FALSE;
				tyP0700LFCtrl.tyMsgBoxTerminateOpsAsk.tyBtnYes.bValue	:= FALSE;

				p_tyC0008MsgBox ACCESS ADR(tyP0700LFCtrl.tyMsgBoxHide);

				usiLFLeaderCtrlStep	:= 3;

			ELSIF tyP0700LFCtrl.tyMsgBoxTerminateOpsAsk.tyBtnNo.bRtCompl = TRUE THEN
				tyP0700LFCtrl.tyMsgBoxTerminateOpsAsk.tyBtnNo.bRtCompl	:= FALSE;
				tyP0700LFCtrl.tyMsgBoxTerminateOpsAsk.tyBtnNo.bValue	:= FALSE;

				p_tyC0008MsgBox ACCESS ADR(tyP0700LFCtrl.tyMsgBoxHide);

				tyP0700LFCtrl.tyLdr.tyBtnChgAll.bValue		:= tyP0700LFCtrl.tyLdr.tyBtnChgAll.bRtCompl;
				tyP0700LFCtrl.tyLdr.tyBtnChgSeqAuto.bValue	:= tyP0700LFCtrl.tyLdr.tyBtnChgSeqAuto.bRtCompl;
				tyP0700LFCtrl.tyLdr.tyBtnChgSeqMnl.bValue	:= tyP0700LFCtrl.tyLdr.tyBtnChgSeqMnl.bRtCompl;
				tyP0700LFCtrl.tyLdr.tyBtnSyncTm.bValue		:= tyP0700LFCtrl.tyLdr.tyBtnSyncTm.bRtCompl;

				usiLFLeaderCtrlStep	:= 2;

			END_IF

			//Display
			tyP0700LFCtrl.tyLdr.tyBitmapChgAll.usiValueIdx		:= BOOL_TO_USINT(tyP0700LFCtrl.tyLdr.tyBtnChgAll.bRtCompl);
			tyP0700LFCtrl.tyLdr.tyBitmapChgSeqAuto.usiValueIdx	:= BOOL_TO_USINT(tyP0700LFCtrl.tyLdr.tyBtnChgSeqAuto.bRtCompl);
			tyP0700LFCtrl.tyLdr.tyBitmapChgSeqMnl.usiValueIdx	:= BOOL_TO_USINT(tyP0700LFCtrl.tyLdr.tyBtnChgSeqMnl.bRtCompl);
			tyP0700LFCtrl.tyLdr.tyBitmapSyncTm.usiValueIdx		:= BOOL_TO_USINT(tyP0700LFCtrl.tyLdr.tyBtnSyncTm.bRtCompl);

		2:	//Processing
			IF tyP0700LFCtrl.tyLdr.tyBtnChgAll.bRtCompl THEN
				eLFLeaderAct	:= LFActChgAllAuto;

				IF p_eLFLeaderStat = LFActChgAllAuto AND (p_eLFLeaderStatus = Done OR p_eLFLeaderStatus = Error) THEN
					usiLFLeaderCtrlStep	:= 3;
				ELSIF tyP0700LFCtrl.tyLdr.tyBtnChgAll.bValue = FALSE THEN
					usiLFLeaderCtrlStep	:= 1;
				END_IF

			ELSIF tyP0700LFCtrl.tyLdr.tyBtnChgSeqAuto.bRtCompl THEN
				eLFLeaderAct	:= LFActChgSeqAuto;

				IF p_tyMcParamCurr.bLFSeqStayActive = FALSE THEN
					IF p_eLFLeaderStat = LFActChgSeqAuto AND (p_eLFLeaderStatus = Done OR p_eLFLeaderStatus = Error) THEN
						usiLFLeaderCtrlStep	:= 3;
					ELSIF tyP0700LFCtrl.tyLdr.tyBtnChgSeqAuto.bValue = FALSE THEN
						usiLFLeaderCtrlStep	:= 1;
					END_IF
				ELSE
					IF p_eLFLeaderStat = LFActChgSeqAuto AND p_eLFLeaderStatus = Error THEN
						usiLFLeaderCtrlStep	:= 4;
					ELSIF tyP0700LFCtrl.tyLdr.tyBtnChgSeqAuto.bValue = FALSE THEN
						usiLFLeaderCtrlStep	:= 1;
					END_IF
				END_IF

			ELSIF tyP0700LFCtrl.tyLdr.tyBtnChgSeqMnl.bRtCompl THEN
				eLFLeaderAct	:= LFActChgSeqMnl;

				IF p_tyMcParamCurr.bLFSeqStayActive = FALSE THEN
					IF p_eLFLeaderStat = LFActChgSeqMnl AND (p_eLFLeaderStatus = Done OR p_eLFLeaderStatus = Error) THEN
						usiLFLeaderCtrlStep	:= 3;
					ELSIF tyP0700LFCtrl.tyLdr.tyBtnChgSeqMnl.bValue = FALSE THEN
						usiLFLeaderCtrlStep	:= 1;
					END_IF
				ELSE
					IF p_eLFLeaderStat = LFActChgSeqMnl AND p_eLFLeaderStatus = Error THEN
						usiLFLeaderCtrlStep	:= 4;
					ELSIF tyP0700LFCtrl.tyLdr.tyBtnChgSeqMnl.bValue = FALSE THEN
						usiLFLeaderCtrlStep	:= 1;
					END_IF
				END_IF

			ELSIF tyP0700LFCtrl.tyLdr.tyBtnSyncTm.bRtCompl THEN
				eLFLeaderAct	:= LFActSyncPLCTm;

				IF p_eLFLeaderStat = LFActSyncPLCTm AND (p_eLFLeaderStatus = Done OR p_eLFLeaderStatus = Error) THEN
					usiLFLeaderCtrlStep	:= 3;
				ELSIF tyP0700LFCtrl.tyLdr.tyBtnSyncTm.bValue = FALSE THEN
					usiLFLeaderCtrlStep	:= 1;
				END_IF

			END_IF

			//Display
			fbLFLeaderCtrlBlinkTm(IN := TRUE);
			IF fbLFLeaderCtrlBlinkTm.Q = TRUE THEN
				fbLFLeaderCtrlBlinkTm(IN := FALSE);

				tyP0700LFCtrl.tyLdr.tyBitmapChgAll.usiValueIdx		:= BOOL_TO_USINT(USINT_TO_BOOL(tyP0700LFCtrl.tyLdr.tyBitmapChgAll.usiValueIdx) XOR tyP0700LFCtrl.tyLdr.tyBtnChgAll.bRtCompl);
				tyP0700LFCtrl.tyLdr.tyBitmapChgSeqAuto.usiValueIdx	:= BOOL_TO_USINT(USINT_TO_BOOL(tyP0700LFCtrl.tyLdr.tyBitmapChgSeqAuto.usiValueIdx) XOR tyP0700LFCtrl.tyLdr.tyBtnChgSeqAuto.bRtCompl);
				tyP0700LFCtrl.tyLdr.tyBitmapChgSeqMnl.usiValueIdx	:= BOOL_TO_USINT(USINT_TO_BOOL(tyP0700LFCtrl.tyLdr.tyBitmapChgSeqMnl.usiValueIdx) XOR tyP0700LFCtrl.tyLdr.tyBtnChgSeqMnl.bRtCompl);
				tyP0700LFCtrl.tyLdr.tyBitmapSyncTm.usiValueIdx		:= BOOL_TO_USINT(USINT_TO_BOOL(tyP0700LFCtrl.tyLdr.tyBitmapSyncTm.usiValueIdx) XOR tyP0700LFCtrl.tyLdr.tyBtnSyncTm.bRtCompl);
			END_IF

		3:	//Complete Reset
			usiLFLeaderCtrlStep	:= 0;

			eLFLeaderAct	:= LFActIdle;

			fbLFLeaderCtrlBlinkTm(IN := FALSE);

			tyP0700LFCtrl.tyLdr.tyBitmapChgAll.usiValueIdx		:= 0;
			tyP0700LFCtrl.tyLdr.tyBitmapChgSeqAuto.usiValueIdx	:= 0;
			tyP0700LFCtrl.tyLdr.tyBitmapChgSeqMnl.usiValueIdx	:= 0;
			tyP0700LFCtrl.tyLdr.tyBitmapSyncTm.usiValueIdx		:= 0;

			tyP0700LFCtrl.tyLdr.tyBtnChgAll.bRtCompl			:= FALSE;
			tyP0700LFCtrl.tyLdr.tyBtnChgSeqAuto.bRtCompl		:= FALSE;
			tyP0700LFCtrl.tyLdr.tyBtnChgSeqMnl.bRtCompl			:= FALSE;
			tyP0700LFCtrl.tyLdr.tyBtnSyncTm.bRtCompl			:= FALSE;

			tyP0700LFCtrl.tyLdr.tyBtnChgAll.bValue				:= FALSE;
			tyP0700LFCtrl.tyLdr.tyBtnChgSeqAuto.bValue			:= FALSE;
			tyP0700LFCtrl.tyLdr.tyBtnChgSeqMnl.bValue			:= FALSE;
			tyP0700LFCtrl.tyLdr.tyBtnSyncTm.bValue				:= FALSE;

		4:
			p_tyC0008MsgBox ACCESS ADR(tyP0700LFCtrl.tyMsgBoxErrorAsk);

			IF tyP0700LFCtrl.tyMsgBoxErrorAsk.tyBtnNo.bRtCompl = TRUE THEN
				tyP0700LFCtrl.tyMsgBoxErrorAsk.tyBtnNo.bRtCompl	:= FALSE;
				tyP0700LFCtrl.tyMsgBoxErrorAsk.tyBtnNo.bValue	:= FALSE;

				p_tyC0008MsgBox ACCESS ADR(tyP0700LFCtrl.tyMsgBoxHide);

				usiLFLeaderCtrlStep	:= 3;

			END_IF

	END_CASE

END_ACTION
```

#### Act_OptP0700Table.st
```iecst
ACTION Act_OptP0700Table:

	//Call Table FB
	fbP0700Table.sVisuNm			:= tyP0700Table.sVisuNm;
	fbP0700Table.udiWorkAreaStartX	:= 17;
	fbP0700Table.udiWorkAreaEndX	:= 594;
	fbP0700Table.udiWorkAreaStartY	:= 94;
	fbP0700Table.udiWorkAreaEndY	:= 445;
	fbP0700Table.udiMinXDist		:= 20;
	fbP0700Table.udiMinYDist		:= 20;
	fbP0700Table.uiSlideScale		:= c_uiP0700TableSize;
	fbP0700Table.iTotalData			:= UDINT_TO_INT(c_diLFClntNum);
	fbP0700Table.iTotalRow			:= c_uiP0700TableSize;
	fbP0700Table(uiSliderStatus 	:= tyP0700LFCtrl.tyLdr.tyTable1List.tyUISlider.uiRtStat , a_tyUIHotspot := tyP0700LFCtrl.tyLdr.tyTable1List.a_tyHotspot , uiTablePos := tyP0700Table.uiTablePos , iSliderPos := tyP0700LFCtrl.tyLdr.tyTable1List.tyUISlider.iValue);

	tyP0700Table.uiSelectedRow		:= fbP0700Table.uiSelectedRow;
	tyP0700Table.bTableActive		:= fbP0700Table.bTableActive;
	tyP0700Table.bSliderActive		:= fbP0700Table.bSliderActive;

	//Table Content
	IF tyP0700Table.bTableActive = TRUE OR tyP0700Table.bSliderActive = TRUE THEN
		FOR i := 1 TO c_uiP0700TableSize DO
			tyP0700LFCtrl.tyLdr.tyTable1List.a_tyStringDataCol0[i].sValue	:= UINT_TO_STRING(tyP0700Table.uiTablePos + i - 1);
		END_FOR
	END_IF

	//Update Status & Current Recipe
	FOR i := 1 TO c_uiP0700TableSize DO
		tyP0700LFCtrl.tyLdr.tyTable1List.a_tyStringDataCol1[i].sValue	:= p_tyLFLeaderFollowerToLeaderTag[tyP0700Table.uiTablePos + i - 1].sMcNm;
		tyP0700LFCtrl.tyLdr.tyTable1List.a_tyStringDataCol2[i].sValue	:= p_tyLFLeaderFollowerToLeaderTag[tyP0700Table.uiTablePos + i - 1].sIPAddr;
		tyP0700LFCtrl.tyLdr.tyTable1List.a_tyStringDataCol4[i].sValue	:= p_tyLFLeaderFollowerToLeaderTag[tyP0700Table.uiTablePos + i - 1].sCurrProdRcp;

		IF p_tyLFLeaderFollowerToLeaderTag[tyP0700Table.uiTablePos + i - 1].sIPAddr = '' THEN
			tyP0700LFCtrl.tyLdr.tyTable1List.a_tyTxtDataCol3[i].usiValueIdx	:= 0;	//Empty
		ELSIF p_tyLFLeaderFollowerToLeaderTag[tyP0700Table.uiTablePos + i - 1].sIPAddr = '0000' THEN
			tyP0700LFCtrl.tyLdr.tyTable1List.a_tyTxtDataCol3[i].usiValueIdx	:= 1;	//Third Party
		ELSIF p_tyMcParamCurr.a_bLFOnline[tyP0700Table.uiTablePos + i - 1] = FALSE THEN
			tyP0700LFCtrl.tyLdr.tyTable1List.a_tyTxtDataCol3[i].usiValueIdx	:= 2;	//Offline
		ELSIF p_tyLFLeaderFollowerToLeaderTag[tyP0700Table.uiTablePos + i - 1].sIPAddr = p_sHWInfoIPAddr THEN
			tyP0700LFCtrl.tyLdr.tyTable1List.a_tyTxtDataCol3[i].usiValueIdx	:= 4;	//Leader
		ELSIF p_tyLFLeaderFollowerToLeaderTag[tyP0700Table.uiTablePos + i - 1].bSectionLeader = TRUE THEN
			tyP0700LFCtrl.tyLdr.tyTable1List.a_tyTxtDataCol3[i].usiValueIdx	:= 5;	//Section Leader
		ELSIF p_tyLFLeaderFollowerInfo[tyP0700Table.uiTablePos + i - 1].bOnline = TRUE THEN
			tyP0700LFCtrl.tyLdr.tyTable1List.a_tyTxtDataCol3[i].usiValueIdx	:= 6;	//Conected
		ELSE
			tyP0700LFCtrl.tyLdr.tyTable1List.a_tyTxtDataCol3[i].usiValueIdx	:= 3;	//Disconnected
		END_IF
	END_FOR

	//Update Color
	FOR i := 1 TO c_uiP0700TableSize DO

		IF tyP0700LFCtrl.tyLdr.tyTable1List.a_tyTxtDataCol3[i].usiValueIdx > 1 THEN
			IF p_tyLFLeaderFollowerInfo[tyP0700Table.uiTablePos + i - 1].bOnline = TRUE THEN
				tyP0700LFCtrl.tyLdr.tyTable1List.a_tyTxtDataCol3[i].usiColor	:= 1;
			ELSE
				tyP0700LFCtrl.tyLdr.tyTable1List.a_tyTxtDataCol3[i].usiColor	:= 2;
			END_IF
		ELSE
			tyP0700LFCtrl.tyLdr.tyTable1List.a_tyTxtDataCol3[i].usiColor	:= 0;
		END_IF

	END_FOR

END_ACTION
```

#### Act_EntP0800Disp.st
```iecst
ACTION Act_EntP0800Disp:

	//Access Address
	p_tyC0005Main ACCESS ADR(tyCommon.tyMain);

	p_tyC0007Notif ACCESS ADR(tyCommon.tyNotif);

	p_tyC0008MsgBox ACCESS ADR(tyP0800MagInfo.tyMsgBoxHide);

	p_tyC0009Info ACCESS ADR(tyCommon.tyInfo);

	p_tyP0800MagInfo1 ACCESS ADR(tyP0800MagInfo.tyMagInfo1);
	p_tyP0800MagInfo2 ACCESS ADR(tyP0800MagInfo.tyMagInfo2);

END_ACTION
```

#### Act_OptP0800Table1.st
```iecst
ACTION Act_OptP0800Table1:

	tyP0800MagInfo.tyMagInfo1.tyTable1List.tyUISlider.iMaxValue	:= DINT_TO_INT(p_tyBuffer1DispBffr.diDispIdxEnd) - (c_uiP0800TableSize - 1);

	//Call Table FB
	fbP0800Table1.sVisuNm				:= tyP0800Table1.sVisuNm;
	fbP0800Table1.udiWorkAreaStartX		:= 15;
	fbP0800Table1.udiWorkAreaEndX		:= 365;
	fbP0800Table1.udiWorkAreaStartY		:= 109;
	fbP0800Table1.udiWorkAreaEndY		:= 429;
	fbP0800Table1.udiMinXDist			:= 20;
	fbP0800Table1.udiMinYDist			:= 20;
	fbP0800Table1.uiSlideScale			:= c_uiP0800TableSize;
	fbP0800Table1.iTotalData			:= DINT_TO_INT(p_tyBuffer1DispBffr.diDispIdxEnd);
	fbP0800Table1.iTotalRow				:= c_uiP0800TableSize;
	fbP0800Table1(uiSliderStatus 		:= tyP0800MagInfo.tyMagInfo1.tyTable1List.tyUISlider.uiRtStat , a_tyUIHotspot := tyP0800MagInfo.tyMagInfo1.tyTable1List.a_tyHotspot , uiTablePos := tyP0800Table1.uiTablePos , iSliderPos := tyP0800MagInfo.tyMagInfo1.tyTable1List.tyUISlider.iValue);

	tyP0800Table1.uiSelectedRow	:= fbP0800Table1.uiSelectedRow;
	tyP0800Table1.bTableActive	:= fbP0800Table1.bTableActive;
	tyP0800Table1.bSliderActive	:= fbP0800Table1.bSliderActive;

	//Table Content
	IF p_tyDI.bMagPresentSen1 THEN
		FOR i := 1 TO c_uiP0800TableSize DO
			tyP0800MagInfo.tyMagInfo1.tyTable1List.a_tyStringDataCol0[i].sValue		:= p_tyBuffer1DispBffr.a_tyDispBffrDat[tyP0800Table1.uiTablePos + i - 1].sSltIdx;
			tyP0800MagInfo.tyMagInfo1.tyTable1List.a_tyStringDataCol1[i].sValue		:= p_tyBuffer1DispBffr.a_tyDispBffrDat[tyP0800Table1.uiTablePos + i - 1].sSltTm;
			tyP0800MagInfo.tyMagInfo1.tyTable1List.a_tyStringDataCol1[i].usiColor	:= DWORD_TO_USINT(p_tyBuffer1DispBffr.a_tyDispBffrDat[tyP0800Table1.uiTablePos + i - 1].dwColor);

		END_FOR
	ELSE
		FOR i := 1 TO c_uiP0800TableSize DO
			tyP0800MagInfo.tyMagInfo1.tyTable1List.a_tyStringDataCol0[i].sValue		:= '';
			tyP0800MagInfo.tyMagInfo1.tyTable1List.a_tyStringDataCol1[i].sValue		:= '';
			tyP0800MagInfo.tyMagInfo1.tyTable1List.a_tyStringDataCol1[i].usiColor	:= 0;

		END_FOR
	END_IF

	tyP0800MagInfo.tyMagInfo1.tyTable1List.tyUISlider.iMaxValue	:= DINT_TO_INT(p_tyBuffer1DispBffr.diDispIdxEnd) - (c_uiP0800TableSize - 1);

END_ACTION
```

#### Act_OptP0800Mag1Updt.st
```iecst
ACTION Act_OptP0800Mag1Updt:

	IF p_tyDI.bMagPresentSen1 THEN
		IF p_tyBuffer1BffrStat.bBffrFull THEN
			tyP0800MagInfo.tyMagInfo1.tyTxtMag1Stat.usiValueIdx	:= 2;
			tyP0800MagInfo.tyMagInfo1.tyTxtMag1Stat.usiColor	:= 1;
		ELSIF p_tyBuffer1BffrStat.bBffrMty THEN
			tyP0800MagInfo.tyMagInfo1.tyTxtMag1Stat.usiValueIdx := 1;
			tyP0800MagInfo.tyMagInfo1.tyTxtMag1Stat.usiColor	:= 0;
		ELSE
			tyP0800MagInfo.tyMagInfo1.tyTxtMag1Stat.usiValueIdx := 3;
			tyP0800MagInfo.tyMagInfo1.tyTxtMag1Stat.usiColor	:= 2;
		END_IF
	ELSE
		tyP0800MagInfo.tyMagInfo1.tyTxtMag1Stat.usiValueIdx		:= 0;
		tyP0800MagInfo.tyMagInfo1.tyTxtMag1Stat.usiColor		:= 1;
	END_IF

	//Set Magazine Full
	IF tyP0800MagInfo.tyMagInfo1.tyBtnMag1SetFull.bRtCompl THEN
		tyP0800MagInfo.tyMagInfo1.tyBtnMag1SetFull.bValue	:= TRUE;

		eBuffer1Act	:= BufferActSetFull;

		IF p_eBuffer1Stat = BufferActSetFull AND p_eBuffer1Status = Done THEN
			eBuffer1Act	:= BufferActIdle;

			tyP0800MagInfo.tyMagInfo1.tyBtnMag1SetFull.bRtCompl	:= FALSE;
			tyP0800MagInfo.tyMagInfo1.tyBtnMag1SetFull.bValue	:= FALSE;
		END_IF
	END_IF

	IF p_bOpsRun THEN
		tyP0800MagInfo.tyMagInfo1.tyBtnMag1SetFull.uiMaskRtStat.0	:= p_tyDI.bMagPresentSen1 AND NOT p_tyBuffer1BffrStat.bBffrFull AND p_bOpsMagConvUL1RlsMagAllw;
	ELSE
		tyP0800MagInfo.tyMagInfo1.tyBtnMag1SetFull.uiMaskRtStat.0	:= p_tyDI.bMagPresentSen1 AND NOT p_tyBuffer1BffrStat.bBffrFull;
	END_IF

END_ACTION
```

#### Act_OptP0800Table2.st
```iecst
ACTION Act_OptP0800Table2:

	tyP0800MagInfo.tyMagInfo1.tyTable2List.tyUISlider.iMaxValue	:= DINT_TO_INT(p_tyBuffer2DispBffr.diDispIdxEnd) - (c_uiP0800TableSize - 1);

	//Call Table FB
	fbP0800Table2.sVisuNm				:= tyP0800Table2.sVisuNm;
	fbP0800Table2.udiWorkAreaStartX		:= 15;
	fbP0800Table2.udiWorkAreaEndX		:= 365;
	fbP0800Table2.udiWorkAreaStartY		:= 109;
	fbP0800Table2.udiWorkAreaEndY		:= 429;
	fbP0800Table2.udiMinXDist			:= 20;
	fbP0800Table2.udiMinYDist			:= 20;
	fbP0800Table2.uiSlideScale			:= c_uiP0800TableSize;
	fbP0800Table2.iTotalData			:= DINT_TO_INT(p_tyBuffer2DispBffr.diDispIdxEnd);
	fbP0800Table2.iTotalRow				:= c_uiP0800TableSize;
	fbP0800Table2(uiSliderStatus 		:= tyP0800MagInfo.tyMagInfo1.tyTable2List.tyUISlider.uiRtStat , a_tyUIHotspot := tyP0800MagInfo.tyMagInfo1.tyTable2List.a_tyHotspot , uiTablePos := tyP0800Table2.uiTablePos , iSliderPos := tyP0800MagInfo.tyMagInfo1.tyTable2List.tyUISlider.iValue);

	tyP0800Table2.uiSelectedRow	:= fbP0800Table2.uiSelectedRow;
	tyP0800Table2.bTableActive	:= fbP0800Table2.bTableActive;
	tyP0800Table2.bSliderActive	:= fbP0800Table2.bSliderActive;

	//Table Content
	IF p_tyDI.bMagPresentSen2 THEN
		FOR i := 1 TO c_uiP0800TableSize DO
			tyP0800MagInfo.tyMagInfo1.tyTable2List.a_tyStringDataCol0[i].sValue		:= p_tyBuffer2DispBffr.a_tyDispBffrDat[tyP0800Table2.uiTablePos + i - 1].sSltIdx;
			tyP0800MagInfo.tyMagInfo1.tyTable2List.a_tyStringDataCol1[i].sValue		:= p_tyBuffer2DispBffr.a_tyDispBffrDat[tyP0800Table2.uiTablePos + i - 1].sSltTm;
			tyP0800MagInfo.tyMagInfo1.tyTable2List.a_tyStringDataCol1[i].usiColor	:= DWORD_TO_USINT(p_tyBuffer2DispBffr.a_tyDispBffrDat[tyP0800Table2.uiTablePos + i - 1].dwColor);

		END_FOR
	ELSE
		FOR i := 1 TO c_uiP0800TableSize DO
			tyP0800MagInfo.tyMagInfo1.tyTable2List.a_tyStringDataCol0[i].sValue		:= '';
			tyP0800MagInfo.tyMagInfo1.tyTable2List.a_tyStringDataCol1[i].sValue		:= '';
			tyP0800MagInfo.tyMagInfo1.tyTable2List.a_tyStringDataCol1[i].usiColor	:= 0;

		END_FOR
	END_IF

	tyP0800MagInfo.tyMagInfo1.tyTable2List.tyUISlider.iMaxValue	:= DINT_TO_INT(p_tyBuffer2DispBffr.diDispIdxEnd) - (c_uiP0800TableSize - 1);

END_ACTION
```

#### Act_OptP0800Mag2Updt.st
```iecst
ACTION Act_OptP0800Mag2Updt:

	IF p_tyDI.bMagPresentSen2 THEN
		IF p_tyBuffer2BffrStat.bBffrFull THEN
			tyP0800MagInfo.tyMagInfo1.tyTxtMag2Stat.usiValueIdx	:= 2;
			tyP0800MagInfo.tyMagInfo1.tyTxtMag2Stat.usiColor	:= 1;
		ELSIF p_tyBuffer2BffrStat.bBffrMty THEN
			tyP0800MagInfo.tyMagInfo1.tyTxtMag2Stat.usiValueIdx := 1;
			tyP0800MagInfo.tyMagInfo1.tyTxtMag2Stat.usiColor	:= 0;
		ELSE
			tyP0800MagInfo.tyMagInfo1.tyTxtMag2Stat.usiValueIdx := 3;
			tyP0800MagInfo.tyMagInfo1.tyTxtMag2Stat.usiColor	:= 2;
		END_IF
	ELSE
		tyP0800MagInfo.tyMagInfo1.tyTxtMag2Stat.usiValueIdx		:= 0;
		tyP0800MagInfo.tyMagInfo1.tyTxtMag2Stat.usiColor		:= 1;
	END_IF

	//Set Magazine Full
	IF tyP0800MagInfo.tyMagInfo1.tyBtnMag2SetFull.bRtCompl THEN
		tyP0800MagInfo.tyMagInfo1.tyBtnMag2SetFull.bValue	:= TRUE;

		eBuffer2Act	:= BufferActSetFull;

		IF p_eBuffer2Stat = BufferActSetFull AND p_eBuffer2Status = Done THEN
			eBuffer2Act	:= BufferActIdle;

			tyP0800MagInfo.tyMagInfo1.tyBtnMag2SetFull.bRtCompl	:= FALSE;
			tyP0800MagInfo.tyMagInfo1.tyBtnMag2SetFull.bValue	:= FALSE;
		END_IF
	END_IF

	IF p_bOpsRun THEN
		tyP0800MagInfo.tyMagInfo1.tyBtnMag2SetFull.uiMaskRtStat.0	:= p_tyDI.bMagPresentSen2 AND NOT p_tyBuffer2BffrStat.bBffrFull AND p_bOpsMagConvUL2RlsMagAllw;
	ELSE
		tyP0800MagInfo.tyMagInfo1.tyBtnMag2SetFull.uiMaskRtStat.0   := p_tyDI.bMagPresentSen2 AND NOT p_tyBuffer2BffrStat.bBffrFull;
	END_IF

END_ACTION
```

#### Act_OptP0800Table3.st
```iecst
ACTION Act_OptP0800Table3:

	tyP0800MagInfo.tyMagInfo2.tyTable3List.tyUISlider.iMaxValue	:= DINT_TO_INT(p_tyBuffer3DispBffr.diDispIdxEnd) - (c_uiP0800TableSize - 1);

	//Call Table FB
	fbP0800Table3.sVisuNm				:= tyP0800Table3.sVisuNm;
	fbP0800Table3.udiWorkAreaStartX		:= 15;
	fbP0800Table3.udiWorkAreaEndX		:= 365;
	fbP0800Table3.udiWorkAreaStartY		:= 109;
	fbP0800Table3.udiWorkAreaEndY		:= 429;
	fbP0800Table3.udiMinXDist			:= 20;
	fbP0800Table3.udiMinYDist			:= 20;
	fbP0800Table3.uiSlideScale			:= c_uiP0800TableSize;
	fbP0800Table3.iTotalData			:= DINT_TO_INT(p_tyBuffer3DispBffr.diDispIdxEnd);
	fbP0800Table3.iTotalRow				:= c_uiP0800TableSize;
	fbP0800Table3(uiSliderStatus 		:= tyP0800MagInfo.tyMagInfo2.tyTable3List.tyUISlider.uiRtStat , a_tyUIHotspot := tyP0800MagInfo.tyMagInfo2.tyTable3List.a_tyHotspot , uiTablePos := tyP0800Table3.uiTablePos , iSliderPos := tyP0800MagInfo.tyMagInfo2.tyTable3List.tyUISlider.iValue);

	tyP0800Table3.uiSelectedRow	:= fbP0800Table3.uiSelectedRow;
	tyP0800Table3.bTableActive	:= fbP0800Table3.bTableActive;
	tyP0800Table3.bSliderActive	:= fbP0800Table3.bSliderActive;

	//Table Content
	IF p_tyDI.bMagPresentSen3 THEN
		FOR i := 1 TO c_uiP0800TableSize DO
			tyP0800MagInfo.tyMagInfo2.tyTable3List.a_tyStringDataCol0[i].sValue		:= p_tyBuffer3DispBffr.a_tyDispBffrDat[tyP0800Table3.uiTablePos + i - 1].sSltIdx;
			tyP0800MagInfo.tyMagInfo2.tyTable3List.a_tyStringDataCol1[i].sValue		:= p_tyBuffer3DispBffr.a_tyDispBffrDat[tyP0800Table3.uiTablePos + i - 1].sSltTm;
			tyP0800MagInfo.tyMagInfo2.tyTable3List.a_tyStringDataCol1[i].usiColor	:= DWORD_TO_USINT(p_tyBuffer3DispBffr.a_tyDispBffrDat[tyP0800Table3.uiTablePos + i - 1].dwColor);

		END_FOR
	ELSE
		FOR i := 1 TO c_uiP0800TableSize DO
			tyP0800MagInfo.tyMagInfo2.tyTable3List.a_tyStringDataCol0[i].sValue		:= '';
			tyP0800MagInfo.tyMagInfo2.tyTable3List.a_tyStringDataCol1[i].sValue		:= '';
			tyP0800MagInfo.tyMagInfo2.tyTable3List.a_tyStringDataCol1[i].usiColor	:= 0;

		END_FOR
	END_IF

	tyP0800MagInfo.tyMagInfo2.tyTable3List.tyUISlider.iMaxValue	:= DINT_TO_INT(p_tyBuffer3DispBffr.diDispIdxEnd) - (c_uiP0800TableSize - 1);

END_ACTION
```

#### Act_OptP0800Mag3Updt.st
```iecst
ACTION Act_OptP0800Mag3Updt:

	IF p_tyDI.bMagPresentSen3 THEN
		IF p_tyBuffer3BffrStat.bBffrFull THEN
			tyP0800MagInfo.tyMagInfo2.tyTxtMag3Stat.usiValueIdx	:= 2;
			tyP0800MagInfo.tyMagInfo2.tyTxtMag3Stat.usiColor	:= 1;
		ELSIF p_tyBuffer3BffrStat.bBffrMty THEN
			tyP0800MagInfo.tyMagInfo2.tyTxtMag3Stat.usiValueIdx := 1;
			tyP0800MagInfo.tyMagInfo2.tyTxtMag3Stat.usiColor	:= 0;
		ELSE
			tyP0800MagInfo.tyMagInfo2.tyTxtMag3Stat.usiValueIdx := 3;
			tyP0800MagInfo.tyMagInfo2.tyTxtMag3Stat.usiColor	:= 2;
		END_IF
	ELSE
		tyP0800MagInfo.tyMagInfo2.tyTxtMag3Stat.usiValueIdx		:= 0;
		tyP0800MagInfo.tyMagInfo2.tyTxtMag3Stat.usiColor		:= 1;
	END_IF

	//Set Magazine Full
	IF tyP0800MagInfo.tyMagInfo2.tyBtnMag3SetFull.bRtCompl THEN
		tyP0800MagInfo.tyMagInfo2.tyBtnMag3SetFull.bValue	:= TRUE;

		eBuffer3Act	:= BufferActSetFull;

		IF p_eBuffer3Stat = BufferActSetFull AND p_eBuffer3Status = Done THEN
			eBuffer3Act	:= BufferActIdle;

			tyP0800MagInfo.tyMagInfo2.tyBtnMag3SetFull.bRtCompl	:= FALSE;
			tyP0800MagInfo.tyMagInfo2.tyBtnMag3SetFull.bValue	:= FALSE;
		END_IF
	END_IF

	IF p_bOpsRun THEN
		tyP0800MagInfo.tyMagInfo2.tyBtnMag3SetFull.uiMaskRtStat.0	:= p_tyDI.bMagPresentSen3 AND NOT p_tyBuffer3BffrStat.bBffrFull AND p_bOpsMagConvUL3RlsMagAllw;
	ELSE
		tyP0800MagInfo.tyMagInfo2.tyBtnMag3SetFull.uiMaskRtStat.0   := p_tyDI.bMagPresentSen3 AND NOT p_tyBuffer3BffrStat.bBffrFull;
	END_IF

END_ACTION
```

#### Act_EntP0850Disp.st
```iecst
ACTION Act_EntP0850Disp:

	//Access Address
	p_tyC0005Main ACCESS ADR(tyCommon.tyMain);

	p_tyC0007Notif ACCESS ADR(tyCommon.tyNotif);

	p_tyC0008MsgBox ACCESS ADR(tyP0850OvenInfo.tyMsgBoxHide);

	p_tyC0009Info ACCESS ADR(tyCommon.tyInfo);

	p_tyP0850OvenCom ACCESS ADR(tyP0850OvenInfo.tyCom);
	p_tyP0850OvenExtddSingle ACCESS ADR(tyP0850OvenInfo.tyExtddA);
	p_tyP0850OvenExtddDualSeparate ACCESS ADR(tyP0850OvenInfo.tyExtddABSeparate);
	p_tyP0850OvenExtddDualMix ACCESS ADR(tyP0850OvenInfo.tyExtddABMix);
	p_tyP0850OvenStdSingle ACCESS ADR(tyP0850OvenInfo.tyStdA);
	p_tyP0850OvenStdDual ACCESS ADR(tyP0850OvenInfo.tyStdAB);

	//Display
	fUIInRtStatHide(ADR(tyP0850OvenInfo.tyStdA.tyLyr.uiRtStat));
	fUIInRtStatHide(ADR(tyP0850OvenInfo.tyStdB.tyLyr.uiRtStat));
	fUIInRtStatHide(ADR(tyP0850OvenInfo.tyStdAB.tyLyr.uiRtStat));

	fUIInRtStatHide(ADR(tyP0850OvenInfo.tyExtddA.tyLyr.uiRtStat));
	fUIInRtStatHide(ADR(tyP0850OvenInfo.tyExtddB.tyLyr.uiRtStat));
	fUIInRtStatHide(ADR(tyP0850OvenInfo.tyExtddABSeparate.tyLyr.uiRtStat));
	fUIInRtStatHide(ADR(tyP0850OvenInfo.tyExtddABMix.tyLyr.uiRtStat));

	IF p_tyNtParamCurr.bOvenInfoExtdPrep = TRUE AND p_tyMcParamCurr.bExtdOvenEn = TRUE THEN
		//Extended Mode
		tyP0850OvenInfo.tyCom.tyTxtTittle.usiValueIdx	:= 1;

		CASE p_tyProdRcpCurrRcp2.usiMcMod OF
			ULModUnloadFrontLnA, ULModRejFrontLnA, ULModRejFrontLnARev:

				fUIInRtStatOff(ADR(tyP0850OvenInfo.tyExtddA.tyLyr.uiRtStat));
				p_tyP0850OvenExtddSingle ACCESS ADR(tyP0850OvenInfo.tyExtddA);

			ULModUnloadRearLnB, ULModRejRearLnB, ULModRejRearLnBRev:

				fUIInRtStatOff(ADR(tyP0850OvenInfo.tyExtddB.tyLyr.uiRtStat));
				p_tyP0850OvenExtddSingle ACCESS ADR(tyP0850OvenInfo.tyExtddB);

			ULModUnloadDualLnAB:

				fUIInRtStatOff(ADR(tyP0850OvenInfo.tyExtddABSeparate.tyLyr.uiRtStat));
				p_tyP0850OvenExtddDualSeparate ACCESS ADR(tyP0850OvenInfo.tyExtddABSeparate);

			ULModRejDualLnA, ULModRejDualLnB:

				fUIInRtStatOff(ADR(tyP0850OvenInfo.tyExtddABMix.tyLyr.uiRtStat));
				p_tyP0850OvenExtddDualMix ACCESS ADR(tyP0850OvenInfo.tyExtddABMix);

		END_CASE

	ELSE
		//Standard Mode
		tyP0850OvenInfo.tyCom.tyTxtTittle.usiValueIdx	:= 0;

		CASE p_tyProdRcpCurrRcp2.usiMcMod OF
			ULModUnloadFrontLnA, ULModRejFrontLnA, ULModRejFrontLnARev:

				p_tyP0850OvenStdSingle ACCESS ADR(tyP0850OvenInfo.tyStdA);
				fUIInRtStatOff(ADR(tyP0850OvenInfo.tyStdA.tyLyr.uiRtStat));

			ULModUnloadRearLnB, ULModRejRearLnB, ULModRejRearLnBRev:

				p_tyP0850OvenStdSingle ACCESS ADR(tyP0850OvenInfo.tyStdB);
				fUIInRtStatOff(ADR(tyP0850OvenInfo.tyStdB.tyLyr.uiRtStat));

			ULModUnloadDualLnAB, ULModRejDualLnA, ULModRejDualLnB:

				p_tyP0850OvenStdDual ACCESS ADR(tyP0850OvenInfo.tyStdAB);
				fUIInRtStatOff(ADR(tyP0850OvenInfo.tyStdAB.tyLyr.uiRtStat));

		END_CASE

	END_IF

	tyP0850OvenInfo.tyCom.tyBtnCntrA.uiRtStat.0	:= NOT(p_tyNtParamCurr.bOvenInfoExtdPrep AND p_tyMcParamCurr.bExtdOvenEn);
	tyP0850OvenInfo.tyCom.tyBtnCntrB.uiRtStat.0	:= NOT(p_tyNtParamCurr.bOvenInfoExtdPrep AND p_tyMcParamCurr.bExtdOvenEn AND p_tyNtParamCurr.bProjLaneBPrep);

END_ACTION
```

#### Act_OptP0850UpdtDat.st
```iecst
ACTION Act_OptP0850UpdtDat:

	//Signal
	tyP0850OvenInfo.tyCom.tyBtnCntrA.bValue	:= p_tyDI.bOvenInfeedSigA;
	tyP0850OvenInfo.tyCom.tyBtnOvenA.bValue	:= p_tyDO.bOvenInfoSigA;
	tyP0850OvenInfo.tyCom.tyBtnCntrB.bValue	:= p_tyDI.bOvenInfeedSigB;
	tyP0850OvenInfo.tyCom.tyBtnOvenB.bValue	:= p_tyDO.bOvenInfoSigB;

	//Buffer Info
	tyP0850OvenInfo.tyStdA.tyNumMinReqFreeBffr.diValue				:= p_tyProdRcpCurrRcp2.diMinReqFreeBffr;
	tyP0850OvenInfo.tyStdB.tyNumMinReqFreeBffr.diValue				:= p_tyProdRcpCurrRcp2.diMinReqFreeBffr;
	tyP0850OvenInfo.tyStdAB.tyNumMinReqFreeBffrA.diValue			:= p_tyProdRcpCurrRcp2.diMinReqFreeBffr;
	tyP0850OvenInfo.tyStdAB.tyNumMinReqFreeBffrB.diValue			:= p_tyProdRcpCurrRcp2.diMinReqFreeBffr;

	tyP0850OvenInfo.tyExtddA.tyNumAddBffr.diValue					:= p_tyMcParamCurr.diOvenMaxBffr;
	tyP0850OvenInfo.tyExtddB.tyNumAddBffr.diValue					:= p_tyMcParamCurr.diOvenMaxBffr;
	tyP0850OvenInfo.tyExtddABSeparate.tyNumAddBffrA.diValue			:= p_tyMcParamCurr.diOvenMaxBffr;
	tyP0850OvenInfo.tyExtddABSeparate.tyNumAddBffrB.diValue			:= p_tyMcParamCurr.diOvenMaxBffr;
	tyP0850OvenInfo.tyExtddABMix.tyNumAddBffrA.diValue				:= p_tyMcParamCurr.diOvenMaxBffr;
	tyP0850OvenInfo.tyExtddABMix.tyNumAddBffrB.diValue				:= p_tyMcParamCurr.diOvenMaxBffr;

	tyP0850OvenInfo.tyStdA.tyNumBffrEmptySlt.diValue				:= p_diBufferMagABffrMtySlt;
	tyP0850OvenInfo.tyStdB.tyNumBffrEmptySlt.diValue				:= p_diBufferMagBBffrMtySlt;
	tyP0850OvenInfo.tyStdAB.tyNumBffrEmptySltA.diValue				:= p_diBufferMagABffrMtySlt;
	tyP0850OvenInfo.tyStdAB.tyNumBffrEmptySltB.diValue				:= p_diBufferMagBBffrMtySlt;

	tyP0850OvenInfo.tyExtddA.tyNumBffrEmptySlt.diValue				:= p_diBufferMagABffrMtySlt;
	tyP0850OvenInfo.tyExtddB.tyNumBffrEmptySlt.diValue				:= p_diBufferMagBBffrMtySlt;
	tyP0850OvenInfo.tyExtddABSeparate.tyNumBffrEmptySltA.diValue	:= p_diBufferMagABffrMtySlt;
	tyP0850OvenInfo.tyExtddABSeparate.tyNumBffrEmptySltB.diValue	:= p_diBufferMagBBffrMtySlt;
	tyP0850OvenInfo.tyExtddABMix.tyNumBffrEmptySlt.diValue			:= p_diBufferMagABffrMtySlt;	//p_diBufferMagBBffrMtySlt

END_ACTION
```

#### Act_OptP0850RBrdInOven.st
```iecst
ACTION Act_OptP0850BrdInOven:

	//Reset Board in Oven
	//A
	IF tyP0850OvenInfo.tyExtddA.tyNumBrdInOven.bRtCompl = TRUE THEN

		diSetBrdInOvenA	:= tyP0850OvenInfo.tyExtddA.tyNumBrdInOven.diValue;
		eOvenInfoAAct	:= OvenInfoActSetBrdInOven;

		IF p_eOvenInfoAStatus = Done AND p_eOvenInfoAStat = OvenInfoActSetBrdInOven THEN
			eOvenInfoAAct	:= OvenInfoActIdle;

			tyP0850OvenInfo.tyExtddA.tyNumBrdInOven.bRtCompl	:= FALSE;
		END_IF

	ELSE
		tyP0850OvenInfo.tyExtddA.tyNumBrdInOven.diValue	:= p_diOvenInfoABrdInOven;

	END_IF

	//B
	IF tyP0850OvenInfo.tyExtddB.tyNumBrdInOven.bRtCompl = TRUE THEN

		diSetBrdInOvenB	:= tyP0850OvenInfo.tyExtddB.tyNumBrdInOven.diValue;
		eOvenInfoBAct	:= OvenInfoActSetBrdInOven;

		IF p_eOvenInfoBStatus = Done AND p_eOvenInfoBStat = OvenInfoActSetBrdInOven THEN
			eOvenInfoBAct	:= OvenInfoActIdle;

			tyP0850OvenInfo.tyExtddB.tyNumBrdInOven.bRtCompl	:= FALSE;
		END_IF

	ELSE
		tyP0850OvenInfo.tyExtddB.tyNumBrdInOven.diValue	:= p_diOvenInfoBBrdInOven;

	END_IF

	//AB Separate
	IF tyP0850OvenInfo.tyExtddABSeparate.tyNumBrdInOvenA.bRtCompl = TRUE THEN

		diSetBrdInOvenA	:= tyP0850OvenInfo.tyExtddABSeparate.tyNumBrdInOvenA.diValue;
		eOvenInfoAAct	:= OvenInfoActSetBrdInOven;

		IF p_eOvenInfoAStatus = Done AND p_eOvenInfoAStat = OvenInfoActSetBrdInOven THEN
			eOvenInfoAAct	:= OvenInfoActIdle;

			tyP0850OvenInfo.tyExtddABSeparate.tyNumBrdInOvenA.bRtCompl	:= FALSE;
		END_IF

	ELSE
		tyP0850OvenInfo.tyExtddABSeparate.tyNumBrdInOvenA.diValue	:= p_diOvenInfoABrdInOven;

	END_IF

	IF tyP0850OvenInfo.tyExtddABSeparate.tyNumBrdInOvenB.bRtCompl = TRUE THEN

		diSetBrdInOvenB	:= tyP0850OvenInfo.tyExtddABSeparate.tyNumBrdInOvenB.diValue;
		eOvenInfoBAct	:= OvenInfoActSetBrdInOven;

		IF p_eOvenInfoBStatus = Done AND p_eOvenInfoBStat = OvenInfoActSetBrdInOven THEN
			eOvenInfoBAct	:= OvenInfoActIdle;

			tyP0850OvenInfo.tyExtddABSeparate.tyNumBrdInOvenB.bRtCompl	:= FALSE;
		END_IF

	ELSE
		tyP0850OvenInfo.tyExtddABSeparate.tyNumBrdInOvenB.diValue	:= p_diOvenInfoBBrdInOven;

	END_IF

	//AB Mix
	IF tyP0850OvenInfo.tyExtddABMix.tyNumBrdInOvenA.bRtCompl = TRUE THEN

		diSetBrdInOvenA	:= tyP0850OvenInfo.tyExtddABMix.tyNumBrdInOvenA.diValue;
		eOvenInfoAAct	:= OvenInfoActSetBrdInOven;

		IF p_eOvenInfoAStatus = Done AND p_eOvenInfoAStat = OvenInfoActSetBrdInOven THEN
			eOvenInfoAAct	:= OvenInfoActIdle;

			tyP0850OvenInfo.tyExtddABMix.tyNumBrdInOvenA.bRtCompl	:= FALSE;
		END_IF

	ELSE
		tyP0850OvenInfo.tyExtddABMix.tyNumBrdInOvenA.diValue	:= p_diOvenInfoABrdInOven;

	END_IF

	IF tyP0850OvenInfo.tyExtddABMix.tyNumBrdInOvenB.bRtCompl = TRUE THEN

		diSetBrdInOvenB	:= tyP0850OvenInfo.tyExtddABMix.tyNumBrdInOvenB.diValue;
		eOvenInfoBAct	:= OvenInfoActSetBrdInOven;

		IF p_eOvenInfoBStatus = Done AND p_eOvenInfoBStat = OvenInfoActSetBrdInOven THEN
			eOvenInfoBAct	:= OvenInfoActIdle;

			tyP0850OvenInfo.tyExtddABMix.tyNumBrdInOvenB.bRtCompl	:= FALSE;
		END_IF

	ELSE
		tyP0850OvenInfo.tyExtddABMix.tyNumBrdInOvenB.diValue	:= p_diOvenInfoBBrdInOven;

	END_IF

END_ACTION
```

#### Act_OptP0850Keypad.st
```iecst
ACTION Act_OptP0850Keypad:

	IF fUIOutRtStatTPIsOpen(ADR(tyP0850OvenInfo.tyExtddA.tyNumBrdInOven.uiRtStat)) THEN
		tyProperty.tyKeypad.tyStringTitle.sKeypadTitle	:= tyP0850OvenInfo.tyExtddA.tyNumBrdInOven.sKeypadTitle;

	ELSIF fUIOutRtStatTPIsOpen(ADR(tyP0850OvenInfo.tyExtddB.tyNumBrdInOven.uiRtStat)) THEN
		tyProperty.tyKeypad.tyStringTitle.sKeypadTitle	:= tyP0850OvenInfo.tyExtddB.tyNumBrdInOven.sKeypadTitle;

	ELSIF fUIOutRtStatTPIsOpen(ADR(tyP0850OvenInfo.tyExtddABSeparate.tyNumBrdInOvenA.uiRtStat)) THEN
		tyProperty.tyKeypad.tyStringTitle.sKeypadTitle	:= tyP0850OvenInfo.tyExtddABSeparate.tyNumBrdInOvenA.sKeypadTitle;

	ELSIF fUIOutRtStatTPIsOpen(ADR(tyP0850OvenInfo.tyExtddABSeparate.tyNumBrdInOvenB.uiRtStat)) THEN
		tyProperty.tyKeypad.tyStringTitle.sKeypadTitle	:= tyP0850OvenInfo.tyExtddABSeparate.tyNumBrdInOvenB.sKeypadTitle;

	ELSIF fUIOutRtStatTPIsOpen(ADR(tyP0850OvenInfo.tyExtddABMix.tyNumBrdInOvenA.uiRtStat)) THEN
		tyProperty.tyKeypad.tyStringTitle.sKeypadTitle	:= tyP0850OvenInfo.tyExtddABMix.tyNumBrdInOvenA.sKeypadTitle;

	ELSIF fUIOutRtStatTPIsOpen(ADR(tyP0850OvenInfo.tyExtddABMix.tyNumBrdInOvenB.uiRtStat)) THEN
		tyProperty.tyKeypad.tyStringTitle.sKeypadTitle	:= tyP0850OvenInfo.tyExtddABMix.tyNumBrdInOvenB.sKeypadTitle;

	ELSE
		tyProperty.tyKeypad.tyStringTitle.sKeypadTitle	:= '';

	END_IF

END_ACTION
```

#### Act_EntP0900Disp.st
```iecst
ACTION Act_EntP0900Disp:

	//Access Address
	p_tyC0005Main ACCESS ADR(tyCommon.tyMain);

	p_tyC0007Notif ACCESS ADR(tyCommon.tyNotif);

	p_tyC0008MsgBox ACCESS ADR(tyP0900GenIn.tyMsgBoxHide);

	p_tyC0009Info ACCESS ADR(tyCommon.tyInfo);

	p_tyP0900GenIn1 ACCESS ADR(tyP0900GenIn.tyGenIn1);
	p_tyP0900GenIn2 ACCESS ADR(tyP0900GenIn.tyGenIn2);
	p_tyP0900GenIn3 ACCESS ADR(tyP0900GenIn.tyGenIn3);

END_ACTION
```

#### Act_OptP0900ReadDI.st
```iecst
ACTION Act_OptP0900ReadDI:

	tyP0900GenIn.tyGenIn1.tyBtnSafetyRly.bValue				:= p_tyDI.bSafetyRlySig;
	tyP0900GenIn.tyGenIn1.tyBtnEStop.bValue					:= p_tyDI.bEStopSig;
	tyP0900GenIn.tyGenIn1.tyBtnCoverSW.bValue				:= p_tyDI.bCoverSWSig;
	tyP0900GenIn.tyGenIn1.tyBtnLifterTimingBeltSen.bValue	:= p_tyDI.bLifterTimingBeltSen;
	tyP0900GenIn.tyGenIn1.tyBtnLifterSafetyLmtSW1.bValue	:= p_tyDI.bLifterSafetyLmtSW1;
	tyP0900GenIn.tyGenIn1.tyBtnLifterSafetyLmtSW2.bValue	:= p_tyDI.bLifterSafetyLmtSW2;
	tyP0900GenIn.tyGenIn1.tyBtnMag1PresentSen.bValue		:= p_tyDI.bMagPresentSen1;
	tyP0900GenIn.tyGenIn1.tyBtnMag2PresentSen.bValue		:= p_tyDI.bMagPresentSen2;
	tyP0900GenIn.tyGenIn1.tyBtnMag3PresentSen.bValue		:= p_tyDI.bMagPresentSen3;
	tyP0900GenIn.tyGenIn1.tyBtnOvenInfeedSigA.bValue		:= p_tyDI.bOvenInfeedSigA;
	tyP0900GenIn.tyGenIn1.tyBtnOvenInfeedSigB.bValue		:= p_tyDI.bOvenInfeedSigB;

	tyP0900GenIn.tyGenIn2.tyBtnMag1OrientationChkSen1.bValue	:= p_tyDI.bMag1OrientChkSen1;
	tyP0900GenIn.tyGenIn2.tyBtnMag1OrientationChkSen2.bValue	:= p_tyDI.bMag1OrientChkSen2;
	tyP0900GenIn.tyGenIn2.tyBtnMag2OrientationChkSen1.bValue	:= p_tyDI.bMag2OrientChkSen1;
	tyP0900GenIn.tyGenIn2.tyBtnMag2OrientationChkSen2.bValue	:= p_tyDI.bMag2OrientChkSen2;
	tyP0900GenIn.tyGenIn2.tyBtnMag3OrientationChkSen1.bValue	:= p_tyDI.bMag3OrientChkSen1;
	tyP0900GenIn.tyGenIn2.tyBtnMag3OrientationChkSen2.bValue	:= p_tyDI.bMag3OrientChkSen2;
	tyP0900GenIn.tyGenIn2.tyBtnMag1HeightSen.bValue				:= p_tyDI.bHighMagDetSen1;
	tyP0900GenIn.tyGenIn2.tyBtnMag2HeightSen.bValue				:= p_tyDI.bHighMagDetSen2;
	tyP0900GenIn.tyGenIn2.tyBtnMag3HeightSen.bValue				:= p_tyDI.bHighMagDetSen3;

	tyP0900GenIn.tyGenIn3.tyBtnCurtainSen.bValue		:= p_tyDI.bCurtainSen;
	tyP0900GenIn.tyGenIn3.tyBtnCurtainSenPB.bValue		:= p_tyDI.bCurtainSenPB;

	tyP0900GenIn.tyGenIn1.tyBtnMagWidthChk.bValue		:= p_tyDI.bMagWidthChkSen;

END_ACTION
```

#### Act_EntP0910Disp.st
```iecst
ACTION Act_EntP0910Disp:

	//Access Address
	p_tyC0005Main ACCESS ADR(tyCommon.tyMain);

	p_tyC0007Notif ACCESS ADR(tyCommon.tyNotif);

	p_tyC0008MsgBox ACCESS ADR(tyP0910GenOut.tyMsgBoxHide);

	p_tyC0009Info ACCESS ADR(tyCommon.tyInfo);

	p_tyP0910GenOut ACCESS ADR(tyP0910GenOut.tyGenOut);
	p_tyP0910GenOutOven ACCESS ADR(tyP0910GenOut.tyOven);
	p_tyP0910MagAW ACCESS ADR(tyP0910GenOut.tyMagAW);
	p_tyP0910GenOutCurtainSen ACCESS ADR(tyP0910GenOut.tyGenOutCurtainSen);

	tyP0910GenOut.tyOven.tyBtnOvenInfoA.uiRtStat.0	:= NOT (p_tyNtParamCurr.bOvenInfoPrep AND p_tyMcParamCurr.bOvenEn );

END_ACTION
```
